(* IEC 61131-3 sources: brOscatLib/oscatNetw (part 3) *)

(* ---- HTTP_GET.st ---- *)
FUNCTION_BLOCK HTTP_GET
    (*http://www.oscat.de/images/OSCATNetwork/oscat_netlib121_en.pdf#page=98*)
    CASE state OF
    00:	DONE := FALSE;
    	IF GET AND NOT get_last THEN (* auf positive Flanke SET warten *)
    		state := 10;
    		ip4_stored := IP4; (* aktuelle IP4 speichern *)
    		total_size := 0;
    		HEADER_START := UINT#0;
    		HEADER_STOP := UINT#0;
    		BODY_START := UINT#0;
    		BODY_STOP := UINT#0;
    		HTTP_STATUS := '';
    		ERROR := DWORD#0;
    		ip_state := BYTE#1; (* Anmelden *)
    		authentication := FALSE;
    		delimiter2b := '$0D$0A';
    		delimiter4b := '$0D$0A$0D$0A';

    		(* LOGIN Parameter vorhanden *)
    		(* LOGIN Parameter vorhanden *)
    		IF URL_DATA.USER <> '' AND URL_DATA.PASSWORD <> '' THEN
    			b64_str1 := CONCAT(URL_DATA.USER,':');
    			b64_str1 := CONCAT(b64_str1,URL_DATA.PASSWORD); (* USER:PASSWORD *)
    			b64_start := TRUE; (* BASE64 kodierung von Username *)
    			authentication := TRUE;
    			state := 5;
    		ELSE
    			state := 10;
    		END_IF
    	        	(*####################  DEBUG-MESSAGE  ###################################*)
    		(*IF _debug_enable THEN
    	       		LOG_CL.NEW_MSG := 'HTTP: S00 START /ip_id ~4';
    	            	LOG_CL.PRINTF[4]  := BYTE_TO_STRING(ip_id);
    	            	LOG_MSG();
    	        	END_IF*)
    	        	(*########################################################################*)
    	END_IF

    5:	IF b64_start AND b64_done THEN (* warten auf base64 konvertierung *)
    		b64_start := FALSE;
    		state := 10;
    	END_IF

    10:	IF ip_state = BYTE#3 THEN (* Bei IP_Control anmelden und auf freigabe warten *)
    		idx := 0;
    		text := CONCAT('GET ',URL_DATA.PATH);
    		_STRING_TO_BUFFER(STR:=text,POS:=idx,PT:=ADR(S_BUF.BUFFER),SIZE:=SIZEOF(S_BUF.BUFFER)); (* GET path in buffer kopieren *)
    		idx := idx + LEN(text);

    		IF LEN(URL_DATA.QUERY) > 0 THEN
    			S_BUF.BUFFER[idx] := 63; (* ASCII '?' *)
    			idx := idx + 1;
    			_STRING_TO_BUFFER(STR:=URL_DATA.QUERY,POS:=idx,PT:=ADR(S_BUF.BUFFER),SIZE:=SIZEOF(S_BUF.BUFFER)); (* QUERY in buffer kopieren *)
    			idx := idx + LEN(URL_DATA.QUERY);
    		END_IF

    		IF MODE >= BYTE#2 THEN (* gewünschte HTTP Version uebergeben *)
    			text := ' HTTP/1.1';
    		ELSE
    			text := ' HTTP/1.0';
    		END_IF
    		text := CONCAT(text,delimiter2b);
    		_STRING_TO_BUFFER(STR:=text,POS:=idx,PT:=ADR(S_BUF.BUFFER),SIZE:=SIZEOF(S_BUF.BUFFER)); (* HTTP Version in buffer kopieren *)
    		idx := idx + LEN(text);

    		IF MODE = BYTE#1 THEN (* HTTP/1.0 mit persistenter Verbindung gewünscht *)
    			text := CONCAT('Connection: Keep-Alive',delimiter2b); (* workaround für pcworx -> kein $0D$0A als Stringkonstante möglich *)
    		ELSIF MODE = BYTE#3 THEN (* HTTP/1.1 ohne persistenter Verbindung gewünscht *)
    			text := CONCAT('Connection: Close',delimiter2b); (* workaround für pcworx -> kein $0D$0A als Stringkonstante möglich *)
    		ELSE
    			text := '';
    		END_IF

    		(* Zusatz Parameter übernehmen *)
    		text := CONCAT(text,URL_DATA.HEADER);
    		_STRING_TO_BUFFER(STR:=text,POS:=idx,PT:=ADR(S_BUF.BUFFER),SIZE:=SIZEOF(S_BUF.BUFFER)); (* HTTP Version in buffer kopieren *)
    		idx := idx + LEN(text);

    		IF authentication THEN
    			text := CONCAT('Authorization: Basic ',b64_str2);
    			text := CONCAT(text,delimiter2b); (* workaround für pcworx -> kein $0D$0A als Stringkonstante möglich *)
    			_STRING_TO_BUFFER(STR:=text,POS:=idx,PT:=ADR(S_BUF.BUFFER),SIZE:=SIZEOF(S_BUF.BUFFER)); (* HTTP Host in buffer kopieren *)
    			idx := idx + LEN(text);
    		END_IF

    		text := CONCAT('Host: ',URL_DATA.DOMAIN);
    		text := CONCAT(text,delimiter4b); (* workaround für pcworx -> kein $0D$0A als Stringkonstante möglich *)
    		_STRING_TO_BUFFER(STR:=text,POS:=idx,PT:=ADR(S_BUF.BUFFER),SIZE:=SIZEOF(S_BUF.BUFFER)); (* HTTP Host in buffer kopieren *)
    		idx := idx + LEN(text);

    		(* IP Datenverkehr einrichten *)
    		IF FIND(';HTTPS;https;Https;', CONCAT(URL_DATA.PROTOCOL,';')) > 1 THEN
    			IP_C.C_PORT := SEL(URL_DATA.PORT = WORD#0,URL_DATA.PORT,WORD#443); (* Portnummer eintragen *)
    			IP_C.MAILBOX[16] := BYTE#1; (* SSL MODE freigeben *)
    		ELSE
    			IP_C.C_PORT := SEL(URL_DATA.PORT = WORD#0,URL_DATA.PORT,WORD#80);  (* Portnummer eintragen *)
    		END_IF

    		IP_C.C_IP := ip4_stored; (* IP eintragen *)
    		IP_C.C_MODE := BYTE#0; (* MODE: TCP+AKTIV+PORT+IP *)
    		IP_C.C_ENABLE := TRUE; (* Verbindungsaufbau freigeben *)
    		IP_C.TIME_RESET := TRUE; (* Zeitueberwachung rücksetzen *)
    		IP_C.R_OBSERVE := TRUE; (* Datenempfang ueberwachen *)
    		S_BUF.SIZE := INT_TO_UINT(idx); (* Sendelänge eintragen *)
    		R_BUF.SIZE := UINT#0; (* Empfangslänge rücksetzen *)

    		state := 30;
    	        	(*####################  DEBUG-MESSAGE  ###################################*)
    	        	(*IF _debug_enable THEN
    	        		LOG_CL.NEW_MSG := 'HTTP: S20 SEND /ip_id ~4';
    	            	LOG_CL.PRINTF[4]  := BYTE_TO_STRING(ip_id);
    	            	LOG_MSG();
    	        	END_IF*)
    	        	(*########################################################################*)
    	END_IF

    30:	rcv_timeout := (IP_C.ERROR AND DWORD#16#0000_FF00) = DWORD#16#0000_FF00;
    	con_rdce :=     (IP_C.ERROR AND DWORD#16#FD00_0000) = DWORD#16#FD00_0000;

    	IF S_BUF.SIZE = UINT#0 THEN
    		IF total_size = 0 THEN
    			IF R_BUF.SIZE > UINT#15 THEN; (* länge der empfangenen Daten prüfen *)

    				(* HTTP HEADER Ende suchen -> durch $0D$A$0D$A erkennbar bei DEC RT-11,CP/M,MS-DOS,Windows *)
    				del_end := '$0D$0A$0D$0A';
    				del_pos := BUFFER_SEARCH(PT:=ADR(R_BUF.BUFFER),SIZE:=R_BUF.SIZE,STR:=del_end,POS:=0,IGN:=FALSE);

    				(* kein Ende gefunden ? -> andere Ende-Codierung suchen *)
    				IF del_pos = 0 THEN
    					del_end := '$0A$0A';
    					(* HTTP HEADER Ende suchen -> durch $0A$0A erkennbar bei Multics, Unix-Derivate,Mac OS X *)
    					del_pos := BUFFER_SEARCH(PT:=ADR(R_BUF.BUFFER),SIZE:=R_BUF.SIZE,STR:=del_end,POS:=0,IGN:=FALSE);
    				END_IF

    				IF del_pos > 0 THEN
    					HEADER_START := UINT#0;
    					HEADER_STOP := INT_TO_UINT(del_pos + LEN(del_end) - 1);
    					total_size := -1; (* HTTP Header empfangen aber noch keine gesamtlänge bekannt *)
    				END_IF
    		                	(*####################  DEBUG-MESSAGE  ###################################*)
    		                	(*IF _debug_enable THEN
    		                   	LOG_CL.NEW_MSG := 'HTTP: S20 HEADER_START ~1 / HEADER_STOP ~2/ip_id ~4';
    		                   	LOG_CL.PRINTF[4]  := BYTE_TO_STRING(ip_id);
    		                   	LOG_CL.PRINTF[1]  := UINT_TO_STRING(HEADER_START);
    		                   	LOG_CL.PRINTF[2]  := UINT_TO_STRING(HEADER_STOP);
    		                   	LOG_MSG();
    		                	END_IF*)
    		                	(*########################################################################*)

    				(* HTTP Statuscode auswerten: (kann 1.0 oder 1.1 sein *)
    				READ_HTTP(size:=HEADER_STOP,pos:=0,SRC:='',pt:=R_BUF.BUFFER);

    				i := LEN(READ_HTTP.READ_HTTP);
    				IF i > 7 THEN
    					(* HTTP Version von HOST auswerten 1.0 oder 1.1 *)
    					text:=MID(READ_HTTP.READ_HTTP,1,3);
    					http_1_1_host := text = '1';

    					(* Code und Meldung isolieren *)
    					HTTP_STATUS := RIGHT(READ_HTTP.READ_HTTP,i-4);
    				END_IF

    				(* positive HTTP Anfrage ? *)
    				IF FIND(HTTP_STATUS,'200') > 0 THEN

    					(* 'Content-Length: Wert einlesen auswerten *)
    					READ_HTTP(size:=HEADER_STOP,pos:=0,SRC:='CONTENT-LENGTH',pt:=R_BUF.BUFFER);
    					text:=READ_HTTP.READ_HTTP;

    					IF LEN(text) >= 1 THEN
    						IF IS_NUM(str:=text) THEN
    							(* erwartete gesamtmenge an Bytes berechnen *)
    							total_size := STRING_TO_INT(text) + UINT_TO_INT(HEADER_STOP) + 1;
                               					(*####################  DEBUG-MESSAGE  ###################################*)
                               					(*IF _debug_enable THEN
                                  					LOG_CL.NEW_MSG := 'HTTP: S20 HEADER ~1, BODY ~2 TOTAL ~3 /ip_id ~4';
                                 					LOG_CL.PRINTF[4]  := BYTE_TO_STRING(ip_id);
                                   					LOG_CL.PRINTF[1]  := UINT_TO_STRING(HEADER_STOP);
                                   					LOG_CL.PRINTF[2]  := INT_TO_STRING(total_size-UINT_TO_INT(HEADER_STOP));
                                   					LOG_CL.PRINTF[3]  := INT_TO_STRING(total_size);
                                  					LOG_MSG();
                              					END_IF*)
                              					(*########################################################################*)
    						END_IF
    					END_IF
    				ELSE
    					ERROR := DWORD#16#000000FC; (* Fehler durch HTTP-Statuscodes *)
    				END_IF
    			END_IF
    		(* 1. bei bekannter Content-Length wird nach erhalt der erwartenen Daten die verbindung beendet *)
    		(* 2. bei persistenter Verbindung muss bei unbekannter Datenmenge auf Receive-Timeout gewartet werden *)
    		(* 3. wenn nach datenempfang die verbindung vom host unterbrochen wird *)
    		ELSIF (R_BUF.SIZE >= INT_TO_UINT(total_size)) OR
    			(R_BUF.SIZE > UINT#0 AND total_size < 0 AND ((rcv_timeout OR con_rdce) OR (IP_C.C_STATE = BYTE#1))) THEN

    			IF R_BUF.SIZE - 1 > HEADER_STOP THEN (* BODY Daten vorhanden *)
    				BODY_START := HEADER_STOP + UINT#1;
    				BODY_STOP := R_BUF.SIZE - 1;
    		                	(*####################  DEBUG-MESSAGE  ###################################*)
    		                	(*IF _debug_enable THEN
    		                   	LOG_CL.NEW_MSG := 'HTTP: S20 BODY ~1, START ~2 END ~3 /ip_id ~4';
    		                   	LOG_CL.PRINTF[4]  := BYTE_TO_STRING(ip_id);
    		                   	LOG_CL.PRINTF[1]  := UINT_TO_STRING(HEADER_STOP);
    		                   	LOG_CL.PRINTF[2]  := UINT_TO_STRING(BODY_START);
    		                   	LOG_CL.PRINTF[3]  := UINT_TO_STRING(BODY_STOP);
    		                   	LOG_MSG();
    		               	END_IF*)
    		               	(*########################################################################*)
    			END_IF

    			DONE := TRUE;
    			IP_C.C_ENABLE := FALSE; (* Verbindung abbauen *)
    			state := 40;
                		(*####################  DEBUG-MESSAGE  ###################################*)
                		(*IF _debug_enable THEN
                    			LOG_CL.NEW_MSG := 'HTTP: S30 OK /ip_id ~4';
                    			LOG_CL.PRINTF[4]  := BYTE_TO_STRING(ip_id);
                    			LOG_MSG();
                		END_IF*)
                		(*########################################################################*)
    		END_IF
    	END_IF

    	IF IP_C.ERROR <> DWORD#0 THEN
    		(* bei unbekannter Content-size ist nicht bekannt ob bzw wieviele Telegramme noch folgen werden *)
    		(* darum wird nach receive-timeout oder Remote disconnect ERROR der fehler wieder ausgefiltert (logischer fehler) *)
    		IF rcv_timeout AND DONE THEN
    			IP_C.ERROR := IP_C.ERROR AND DWORD#16#FFFF_00FF; (* Fehler wieder rücksetzen *)
    		ELSIF con_rdce AND DONE THEN
    			IP_C.ERROR := IP_C.ERROR AND DWORD#16#00FF_FFFF; (* Fehler wieder rücksetzen *)
    		ELSE
    			ERROR := IP_C.ERROR;
    		END_IF
    	END_IF

    	IF ERROR > DWORD#0 THEN
    		IP_C.C_ENABLE := FALSE; (* Verbindungsaufbau sperren *)
    		state := 40;
    	        	(*####################  DEBUG-MESSAGE  ###################################*)
    	        	(*IF _debug_enable THEN
    	            	LOG_CL.NEW_MSG := 'HTTP: S30 ERROR ~1 /ip_id ~4';
    	            	LOG_CL.PRINTF[1]  := DWORD_TO_STRING(ERROR);
    	            	LOG_CL.PRINTF[4]  := BYTE_TO_STRING(ip_id);
    	            	LOG_MSG();
    	        	END_IF*)
    	        	(*########################################################################*)
    	END_IF

    40:	IF (UNLOCK_BUF OR NOT DONE) THEN (* Warten auf Release und Verbindung beendet -> ip_id vom Stack nehmen *)
    		ip_state := BYTE#4; (* Abmelden *)
    		DONE := FALSE;
    		IP_C.MAILBOX[16] := BYTE#0; (* SSL MODE beenden *)
    		state := 0;
    	END_IF
    END_CASE

    get_last := GET; (* letzten Status sichern zur Flankenerkennung *)

    IP_FIFO(FIFO:=IP_C.FIFO,state:=ip_state,ID:=ip_id); (* IP_FIFO *)

    BASE64_ENCODE_STR(RUN:=b64_start,STR1:=b64_str1,STR2:=b64_str2); (* BASE64 kodierung *)
    b64_done:=BASE64_ENCODE_STR.DONE;

    (*####################  DEBUG-MESSAGE  ###################################*)
    (*IF _debug_enable THEN
    	IF state <> _debug_state_last THEN
    		LOG_CL.NEW_MSG := 'http_get: /last ~1 /New ~2';
    		LOG_CL.PRINTF[1] := INT_TO_STRING(_debug_state_last);
    		LOG_CL.PRINTF[2] := INT_TO_STRING(state);
    		LOG_MSG();
    		_debug_state_last := state;
    	END_IF
    END_IF*)
    (*########################################################################*)

    (* revision history
    ks	18. oct. 2008	rev 1.0
    	original version

    ks	20. oct. 2009	rev 1.1
    	Fehler bei body-suche bei $0a$0a korrigiert,Codeoptimierung,
    	new VAR del_pos , del_end (Networkbuffer und Buffer-funktionen auf Basis 0)

    ks	28. oct. 2009	rev 1.2
    	über url.header können zusätzliche header-infos übergeben werden

    ks	12. apr. 2011	rev 1.3
    	verbesserte fehlererkennung und fehlerkorrektur bei buffer_to_string

    ks	31. mar. 2016	rev 1.4
    	authentication und SSL (HTTPS) hinzugefügt, DONE später zurücksetzen

    *)
END_FUNCTION_BLOCK

(* ---- INI_PARSER_BUF.st ---- *)
FUNCTION_BLOCK INI_PARSER_BUF
    (*http://www.oscat.de/images/OSCATNetwork/oscat_netlib121_en.pdf#page=161*)
    IF RUN > 0 THEN
    	IF state = 0 THEN (* Auswertung neu beginnen *)

    		pv := ADR(VALUE);
    		pv := 0; (* VALUE = '' *)
    		pve := pv + INT_TO_DWORD(STRING_LENGTH);
    		pk := ADR(KEY);
    		pk := 0; (* KEY = '' *)
    		pke := pk + INT_TO_DWORD(STRING_LENGTH);

    		i := UDINT_TO_INT(OFFSET);
    		size := UINT_TO_INT(PT.size) - 1;
    		RESULT := 0;
    		state := 5; (* Befehl in Arbeit (Busy) *)
    		step := 0; (* Auswertung neu beginnen *)

    		(*####################  DEBUG-MESSAGE  ###################################*)
    		(*IF _debug_enable THEN
    			LOG_CL.NEW_MSG := 'IPB: Startindex: ~1';
    			LOG_CL.PRINTF[1]  := INT_TO_STRING(i);
    			LOG_MSG();
    		END_IF*)
    		(*########################################################################*)
    	END_IF

    	watchdog(IN:=FALSE,PT:=T#1ms); (* Timer neustarten *)
    	watchdog.IN := TRUE;

    	WHILE (state = 5) DO (* Schleife solange kein Ergebnis *)

    		watchdog(); (* Timer aktualisieren *)

    		IF watchdog.Q THEN (* watchdog ausgelöst *)
    			state := 5;
    			EXIT;
    		ELSIF i > size THEN (* kein weiteres zeichen vorhanden *)
    			state := 10; (* nichts gefunden - Daten-Ende erreicht *)
    			EXIT;
    		ELSE

    			c := PT.BUFFER[i]; (* neues Zeichen aus Buffer lesen *)
    			eof := i + 1 = PT.size; (* End of File *)

    			k_add := 0;
    			v_add := 0;

    			CASE step OF

    			0: (* noch kein Modus erkannt *)
    				IF c = 91 THEN (* mit "[" vergleichen *)
    					step := 200; (* Modus für Section aktivieren *)
    				ELSIF c = 59 OR c = 35 THEN (* mit ";" und '#' vergleichen *)
    					step := 100; (* Modus für Kommentar aktivieren *)
    				ELSIF c > 32 THEN (* KEY erkannt *)
    					k_add := c; (* Zeichen ablegen *)
    					step := 300; (* KEY auswertung starten *)
    				END_IF
    			100: (* Kommentar erkannt -> Zeilenende suchen *)
    				IF c < 32 THEN (* prüfe auf Steuerzeichen *)
    					state  := 3; (* Beenden -> Kommentar wurde gefunden *)
    				END_IF
    			200: (* Sections-start erkannt -> Sectionsende suchen *)
    				IF c = 93 THEN (* mit "]" vergleichen *)
    					IF pk > ADR(KEY) > 0 THEN (* innerhalb von [] muss sich mindestens ein Zeichen befinden *)
    						state  := 1; (* Beenden -> Section wurde gefunden *)
    					ELSE
    						pk := ADR(KEY);
    						pk := 0; (* KEY = '' *)
    						step := 0; (* fehlerhafte Section-Zeile vorhanden -> weitersuchen *)
    					END_IF
    				ELSIF c < 32 OR eof THEN (* Steuerzeichen - fehlerhafte Section-Zeile -> weitersuchen *)
    					pk := ADR(KEY);
    					pk := 0; (* KEY = '' *)
    					step := 0;
    				ELSE
    					k_add := c; (* Zeichen ablegen *)
    				END_IF
    			300: (* Beginn: KEY erkannt -> Name auswerten *)
    				IF c < 32 THEN (* Steuerzeichen - fehlerhafte KEY-Zeile -> weitersuchen *)
    					pk := ADR(KEY);
    					pk := 0; (* KEY = '' *)
    					step := 0;
    				ELSIF c = 61 THEN (* prüfe auf '=' *)
    					step := 330;
    				ELSE
    					k_add := c; (* Zeichen ablegen *)
    				END_IF
    			330: (* KeyValue beginn suchen *)
    				IF c < 32 THEN (* Steuerzeichen  *)
    					state := 2; (* KEY ohne VALUE gefunden *)
    				ELSIF eof THEN
    					state := 2; (* KEY ohne VALUE gefunden *)
    					v_add := c; (* Zeichen ablegen *)
    				ELSE
    					v_add := c; (* Zeichen ablegen *)
    					step := 350;
    				END_IF
    			350: (* KeyValue Ende suchen *)
    				IF c < 32 THEN (* Steuerzeichen *)
    					state := 2; (* KEY gefunden *)
    				ELSIF eof THEN
    					v_add := c; (* Zeichen ablegen *)
    					state := 2; (* KEY gefunden *)
    				ELSE
    					v_add := c; (* Zeichen ablegen *)
    				END_IF
    			END_CASE

    			IF v_add > 0  AND pv < pve THEN (* Zeichen zu VALUE-String hinzufügen *)
    				pv := v_add; (* Zeichen eintragen *)
    				pv := pv + 1;
    				pv := 0; (* String-Terminierung eintragen *)
    			END_IF

    			IF k_add > 0 AND pk < pke THEN (* Zeichen zu KEY-String hinzufügen *)
    				pk := k_add; (* Zeichen eintragen *)
    				pk := pk + 1;
    				pk := 0; (* String-Terminierung eintragen *)
    			END_IF

    			i := i + 1; (* Datenzeiger erhöhen *)

    		END_IF
    	END_WHILE

    	CASE state OF
    	01:	(* Section gefunden *)
    		IF RUN = 1 OR RUN = 3 THEN (* Section vorgewählt oder alles rückmelden *)
    			IF KEY = STR OR LEN(STR) = 0 THEN (* mit gesuchter Section vergleichen oder keine Section vorgegeben *)
    				RESULT := 1; (* Section gefunden *)
    				OFFSET := i; (* OFFSET uebernehmen *)
    				RUN := 0;
    				state := 0;
    			END_IF
    		ELSE
    			pk := ADR(KEY);
    			pk := 0; (* KEY = '' *)
    			RESULT := 11; (* KEY nicht gefunden , Section-Ende - OFFSET nicht verändern *)
    			RUN := 0;
    			state := 0;
    		END_IF
    	02:	(* KEY gefunden *)
    		IF RUN = 2 OR RUN = 3 THEN (* KEY vorgewählt oder alles rückmelden *)
    			IF KEY = STR OR LEN(STR) = 0 THEN (* mit gesuchten KEY vergleichen *)
    				RESULT := 2; (* KEY gefunden *)
    				OFFSET := i; (* OFFSET uebernehmen *)
    				RUN := 0;
    				state := 0;
    			END_IF
    		END_IF
    	03:	(* Kommenar gefunden *)
    		OFFSET := i; (* OFFSET uebernehmen *)
    		state := 0;

    	05:	RESULT := 5; (* in Arbeit *)

    	10:	(* Indexüberschreitung - Bufferende *)
    		RESULT := 10; (* nichts gefunden - Datenende erreicht *)
    		OFFSET := i; (* OFFSET uebernehmen *)
    		RUN := 0;
    		state := 0;
    	END_CASE

    	(*####################  DEBUG-MESSAGE  ###################################*)
    	(*IF _debug_enable THEN
    		LOG_CL.NEW_MSG := 'IPF: intern RESULT ~1 , state ~2, step ~3 , OFFSET ~4, RUN ~5';
    		LOG_CL.PRINTF[1] := BYTE_TO_STRING(RESULT);
    		LOG_CL.PRINTF[2] := BYTE_TO_STRING(state);
    		LOG_CL.PRINTF[3] := INT_TO_STRING(step);
    		LOG_CL.PRINTF[4] := UDINT_TO_STRING(OFFSET);
    		LOG_CL.PRINTF[5] := BYTE_TO_STRING(RUN);
    		LOG_MSG();
    	END_IF*)
    	(*########################################################################*)

    END_IF

    (*####################  DEBUG-MESSAGE  ###################################*)
    (*IF _debug_enable THEN
    	IF step_last <> step THEN
    		LOG_CL.NEW_MSG := 'IPB: step: ~1';
    		LOG_CL.PRINTF[1]  := INT_TO_STRING(step);
    		LOG_MSG();
    	END_IF
    	step_last := step;
    END_IF*)
    (*########################################################################*)

    (* revision history
    ks	23. sep. 2010	rev 1.0
    	original version
    *)
END_FUNCTION_BLOCK

(* ---- INI_PARSER_FILE.st ---- *)
FUNCTION_BLOCK INI_PARSER_FILE
    (*http://www.oscat.de/images/OSCATNetwork/oscat_netlib121_en.pdf#page=164*)
    IF RUN > 0 THEN

    	IF state = 0 THEN (* Auswertung neu beginnen *)
    		pv := ADR(VALUE);
    		pv := 0; (* VALUE = '' *)
    		pve := pv + INT_TO_DWORD(STRING_LENGTH);
    		pk := ADR(KEY);
    		pk := 0; (* KEY = '' *)
    		pke := pk + INT_TO_DWORD(STRING_LENGTH);

    		i := OFFSET;
    		RESULT := 0;
    		state := 5; (* Befehl in Arbeit (Busy) *)
    		step := 0; (* Auswertung neu beginnen *)

    		(*####################  DEBUG-MESSAGE  ###################################*)
    		(*IF _debug_enable THEN
    			LOG_CL.NEW_MSG := 'IPF: Startindex: ~1';
    			LOG_CL.PRINTF[1] := UDINT_TO_STRING(i);
    			LOG_MSG();
    		END_IF*)
    		(*########################################################################*)

    	END_IF

    	watchdog(IN:=FALSE,PT:=T#1ms); (* Timer neustarten *)
    	watchdog.IN := TRUE;

    	WHILE (state = 5) DO (* Schleife solange kein Ergebnis *)

    		mode := 1;
    		FB(mode:=mode,FSD:=FSD,PT:=PT,FILENAME:=FILENAME,POS:=i );
    		e:=FB.ERROR;
    		c:=FB.DATA;

    		eof := i + 1 = FSD.FILE_SIZE; (* End of File *)

    		(*####################  DEBUG-MESSAGE  ###################################*)
    		(*IF _debug_enable THEN
    			LOG_CL.NEW_MSG := 'IPF: mode: ~1, error: ~2 , >~7<>~3< ~4 step ~5 index ~6';
    			LOG_CL.PRINTF[1] := BYTE_TO_STRING(mode);
    			LOG_CL.PRINTF[2] := BYTE_TO_STRING(e);
    			LOG_CL.PRINTF[3] := BYTE_TO_STRING(c);
    			LOG_CL.PRINTF[4] := BOOL_TO_STRING(eof);
    			LOG_CL.PRINTF[5] := INT_TO_STRING(step);
    			LOG_CL.PRINTF[6] := UDINT_TO_STRING(i);
    			LOG_CL.PRINTF[7] := CHR_TO_STRING(c);
    			LOG_MSG();
    		END_IF*)
    		(*########################################################################*)

    		watchdog(); (* Timer aktualisieren *)

    		IF mode > 0 OR watchdog.Q THEN (* Baustein noch aktiv, oder watchdog ausgelöst *)
    			state := 5;
    			EXIT;
    		ELSIF e > 0 THEN (* File_error oder kein weiteres zeichen vorhanden *)
    			state := 10; (* nichts gefunden - Daten-Ende erreicht *)
    			EXIT;
    		ELSE

    			k_add := 0;
    			v_add := 0;

    			CASE step OF

    			0: (* noch kein Modus erkannt *)
    				IF c = 91 THEN (* mit "[" vergleichen *)
    					step := 200; (* Modus für Section aktivieren *)
    				ELSIF c = 59 OR c = 35 THEN (* mit ";" und '#' vergleichen *)
    					step := 100; (* Modus für Kommentar aktivieren *)
    				ELSIF c > 32 THEN (* KEY erkannt *)
    					k_add := c; (* Zeichen ablegen *)
    					step := 300; (* KEY auswertung starten *)
    				END_IF
    			100: (* Kommentar erkannt -> Zeilenende suchen *)
    				IF c < 32 THEN (* prüfe auf Steuerzeichen *)
    					state  := 3; (* Beenden -> Kommentar wurde gefunden *)
    				END_IF
    			200: (* Sections-start erkannt -> Sectionsende suchen *)
    				IF c = 93 THEN (* mit "]" vergleichen *)
    					IF pk > ADR(KEY) > 0 THEN (* innerhalb von [] muss sich mindestens ein Zeichen befinden *)
    						state  := 1; (* Beenden -> Section wurde gefunden *)
    					ELSE
    						pk := ADR(KEY);
    						pk := 0; (* KEY = '' *)
    						step := 0; (* fehlerhafte Section-Zeile vorhanden -> weitersuchen *)
    					END_IF
    				ELSIF c < 32 OR eof THEN (* Steuerzeichen - fehlerhafte Section-Zeile -> weitersuchen *)
    					pk := ADR(KEY);
    					pk := 0; (* KEY = '' *)
    					step := 0;
    				ELSE
    					k_add := c; (* Zeichen ablegen *)
    				END_IF
    			300: (* Beginn: KEY erkannt -> Name auswerten *)
    				IF c < 32 THEN (* Steuerzeichen - fehlerhafte KEY-Zeile -> weitersuchen *)
    					pk := ADR(KEY);
    					pk := 0; (* KEY = '' *)
    					step := 0;
    				ELSIF c = 61 THEN (* prüfe auf '=' *)
    					step := 330;
    				ELSE
    					k_add := c; (* Zeichen ablegen *)
    				END_IF
    			330: (* KeyValue beginn suchen *)
    				IF c < 32 THEN (* Steuerzeichen  *)
    					state := 2; (* KEY ohne VALUE gefunden *)
    				ELSIF eof THEN
    					state := 2; (* KEY ohne VALUE gefunden *)
    					v_add := c; (* Zeichen ablegen *)
    				ELSE
    					v_add := c; (* Zeichen ablegen *)
    					step := 350;
    				END_IF
    			350: (* KeyValue Ende suchen *)
    				IF c < 32 THEN (* Steuerzeichen *)
    					state := 2; (* KEY gefunden *)
    				ELSIF eof THEN
    					v_add := c; (* Zeichen ablegen *)
    					state := 2; (* KEY gefunden *)
    				ELSE
    					v_add := c; (* Zeichen ablegen *)
    				END_IF
    			END_CASE

    			IF v_add > 0  AND pv < pve THEN (* Zeichen zu VALUE-String hinzufügen *)
    				pv := v_add; (* Zeichen eintragen *)
    				pv := pv + 1;
    				pv := 0; (* String-Terminierung eintragen *)
    			END_IF

    			IF k_add > 0 AND pk < pke THEN (* Zeichen zu KEY-String hinzufügen *)
    				pk := k_add; (* Zeichen eintragen *)
    				pk := pk + 1;
    				pk := 0; (* String-Terminierung eintragen *)
    			END_IF

    			i := i + 1; (* Datenzeiger erhöhen *)

    		END_IF
    	END_WHILE

    	CASE state OF
    	01:	(* Section gefunden *)
    		IF RUN = 1 OR RUN = 3 THEN (* Section vorgewählt oder alles rückmelden *)
    			IF KEY = STR OR LEN(STR) = 0 THEN (* mit gesuchter Section vergleichen oder keine Section vorgegeben *)
    				RESULT := 1; (* Section gefunden *)
    				OFFSET := i; (* OFFSET uebernehmen *)
    				RUN := 0;
    				state := 0;
    			END_IF
    		ELSE
    			pk := ADR(KEY);
    			pk := 0; (* KEY = '' *)
    			RESULT := 11; (* KEY nicht gefunden , Section-Ende - OFFSET nicht verändern *)
    			RUN := 0;
    			state := 0;
    		END_IF
    	02:	(* KEY gefunden *)
    		IF RUN = 2 OR RUN = 3 THEN (* KEY vorgewählt oder alles rückmelden *)
    			IF KEY = STR OR LEN(STR) = 0 THEN (* mit gesuchten KEY vergleichen *)
    				RESULT := 2; (* KEY gefunden *)
    				OFFSET := i; (* OFFSET uebernehmen *)
    				RUN := 0;
    				state := 0;
    			END_IF
    		END_IF
    	03:	(* Kommenar gefunden *)
    		OFFSET := i; (* OFFSET uebernehmen *)
    		state := 0;

    	05:	RESULT := 5; (* in Arbeit *)

    	10:	(* Indexüberschreitung - Bufferende *)
    		RESULT := 10; (* nichts gefunden - Datenende erreicht *)
    		OFFSET := i; (* OFFSET uebernehmen *)
    		RUN := 0;
    		state := 0;
    	END_CASE

    	(*####################  DEBUG-MESSAGE  ###################################*)
    	(*IF _debug_enable THEN
    		LOG_CL.NEW_MSG := 'IPF: intern RESULT ~1 , state ~2, step ~3 , OFFSET ~4, RUN ~5';
    		LOG_CL.PRINTF[1] := BYTE_TO_STRING(RESULT);
    		LOG_CL.PRINTF[2] := BYTE_TO_STRING(state);
    		LOG_CL.PRINTF[3] := INT_TO_STRING(step);
    		LOG_CL.PRINTF[4] := UDINT_TO_STRING(OFFSET);
    		LOG_CL.PRINTF[5] := BYTE_TO_STRING(RUN);
    		LOG_MSG();
    	END_IF*)
    	(*########################################################################*)

    END_IF

    (*####################  DEBUG-MESSAGE  ###################################*)
    (*IF _debug_enable THEN
    	IF step_last <> step THEN
    		LOG_CL.NEW_MSG := 'IPB: step: ~1';
    		LOG_CL.PRINTF[1]  := INT_TO_STRING(step);
    		LOG_MSG();
    	END_IF
    	step_last := step;
    END_IF*)
    (*########################################################################*)

    (* revision history
    ks	23. sep. 2010	rev 1.0
    	original version
    *)
END_FUNCTION_BLOCK

(* ---- IP2GEO.st ---- *)
FUNCTION_BLOCK IP2GEO
    (*http://www.oscat.de/images/OSCATNetwork/oscat_netlib121_en.pdf#page=99*)
    CASE state OF

    00:
    	IF ACTIVATE AND NOT last_state THEN
    		state := 20;
    		DONE := FALSE;
    		BUSY := TRUE;
    		ERROR_C := DWORD#0;
    		ERROR_T := BYTE#0;
    	END_IF

    20: (* URL for DNS UND HTTP-GET *)
    	(* Example: http://ipinfodb.com/ip_query.php?IP=10.10.10.10 *)
    	(* Example: http://ipinfodb.com/ip_query.php?timezone=true&IP=*)
    	URL_DATA:=STRING_TO_URL(STR:='http://ipinfodb.com/ip_query.php?timezone=true&IP=',DEFAULT_PROTOCOL:='',DEFAULT_PATH:='');

    	IF IP > DWORD#0 THEN
    		URL_DATA.QUERY := CONCAT(URL_DATA.QUERY,IP4_TO_STRING(IP4:=IP));
    	END_IF

    	state := 40;

    40:
    	IF DNS_CLIENT.DONE THEN
    		state := 60;
    	ELSIF (DNS_CLIENT.ERROR > DWORD#00) THEN
    		(* Fehlerbehandlung *)
    		ERROR_C := DNS_CLIENT.ERROR;
    		ERROR_T := BYTE#01;
    		state := 100;
    	END_IF

    60:
    	IF HTTP_GET.DONE THEN
    		state := 80;
    		CTRL.START_POS := HTTP_GET.BODY_START;
    		CTRL.STOP_POS := HTTP_GET.BODY_STOP;
    		CTRL.COMMAND := WORD#2#10000000_00011000; (* ONLY TEXT AND ATTRIBUTE *)
    		CTRL.WATCHDOG := T#1ms;

    	ELSIF (HTTP_GET.ERROR > DWORD#00) THEN
    		(* Fehlerbehandlung *)
    		ERROR_C := HTTP_GET.ERROR;
    		ERROR_T := BYTE#02;
    		state := 100;
    	END_IF

    80:
    	(* XML Daten seriell lesen *)
    	XML_READER(CTRL:=CTRL,BUF:=R_BUF.BUFFER);
    	IF CTRL.TYP < 98 THEN (* nur auswerten wenn kein Watchdog durchlauf *)
    		(* automatische konvertierung in real und int ausführen *)
    		value_int := 0;
    		value_real := 0.0;
    		IF LEN(CTRL.VALUE) <= 20 THEN
    			v_real :=FLOAT_TO_REAL(FLT:=CTRL.VALUE);
    			IF CHK_REAL(v_real) = 0 THEN (* !!! prüft auf gültigen REAL Wert, ansonsten stürzt Twincat ab !!!!  *)
    				value_real := v_real;
    				value_int := REAL_TO_INT(value_real);
    			END_IF
    		END_IF

    		CASE UINT_TO_INT(CTRL.COUNT) OF

    		07: GEO.IP4 := IP4_DECODE(STR:=CTRL.VALUE); (* IP-Adresse *)
    		10: GEO.state := 'OK' = CTRL.VALUE; (* STATUS *)
    		13: GEO.COUNTRY_CODE := CTRL.VALUE; (* Country-Code *)
    		16: GEO.COUNTRY_NAME := CTRL.VALUE; (* Country-Name *)
    		19: GEO.REGION_CODE := CTRL.VALUE; (* Region-Code *)
    		22: GEO.REGION_NAME := CTRL.VALUE; (* Region-Name *)
    		25: GEO.CITY := CTRL.VALUE; (* City *)
    		31: GEO.GEO_LATITUDE := value_real; (* Latitude *)
    		34: GEO.GEO_LONGITUDE := value_real; (* Longitude *)
    		37: GEO.TIME_ZONE_NAME := CTRL.VALUE; (* TimeZone Name *)
    		40: GEO.GMT_OFFSET := value_int; (* GMT OFFSET in Sekunden *)
    		43: GEO.IS_DST := value_int > 0; (* Sommerzeit aktiv *)
    		END_CASE

    	ELSIF CTRL.TYP = 99 THEN (* EXIT - letztes Element gelesen *)
    		DONE := TRUE;
    		state := 100;
    	END_IF

    100:
    	(* UNLOCK HTTP DATA *)
    	IF (NOT HTTP_GET.DONE) THEN
    		state := 0;
    		BUSY := FALSE;
    		DONE := ERROR_T = BYTE#0;
    	END_IF

    END_CASE

    (* ---------------- DNS --------------- *)
    DNS_CLIENT(	IP_C:=IP_C,
    			S_BUF:=S_BUF,
    			R_BUF:=R_BUF,
    			DOMAIN:=URL_DATA.DOMAIN,
    			IP4_DNS:=DWORD#00,
    			ACTIVATE:=state=40 (* DNS Start *)
    			);

    (* nicht oder nicht direkt verwendete Parameter *)
    (* 	DWORD :=DNS_CLIENT.IP4;
    	BOOL  :=DNS_CLIENT.DONE;
    	BYTE  :=DNS_CLIENT.ERROR; *)
    (* -------------------------------------*)

    (* ------------- HTTP_GET --------------- *)
    HTTP_GET(	IP_C:=IP_C,
    			S_BUF:=S_BUF,
    			R_BUF:=R_BUF,
    			IP4:=DNS_CLIENT.IP4,
    			GET:=state=60,
    			MODE:=BYTE#2, (* HTTP 1.1 mit persistenter Verbindung *)
    			UNLOCK_BUF:=state=100,
    			URL_DATA:=URL_DATA
    			);

    (* nicht oder nicht direkt verwendete Parameter *)
    (*	STRING := HTTP_GET.HTTP_STATUS;
    	UINT :=HTTP_GET.HEADER_START;
    	UINT :=HTTP_GET.HEADER_STOP;
    	UINT :=HTTP_GET.BODY_START;
    	UINT :=HTTP_GET.BODY_STOP;
    	BOOL :=HTTP_GET.DONE;
    	BYTE :=HTTP_GET.ERROR;
    *)
    (* -------------------------------------*)

    last_state := ACTIVATE;

    (* revision history
    ks	14. aug. 2009	rev 1.0
    	original version

    ks	07. oct. 2010	rev 1.1
    	new url , ip2geo fields , REAL_CHECK
    *)
END_FUNCTION_BLOCK

(* ---- IP_CONTROL.st ---- *)
FUNCTION_BLOCK IP_CONTROL
    (*http://www.oscat.de/images/OSCATNetwork/oscat_netlib121_en.pdf#page=101*)
    (* ---------------------- Debug-Message ----------------------------*)
    (*IF _debug_enable THEN
    	IF IP_C.FIFO.ID > BYTE#0 THEN
    		debug_index := IP_C.FIFO.NR;
    		debug_ID := BYTE_TO_INT(IP_C.FIFO.X[debug_index]);
    	END_IF
    END_IF*)
    (* -----------------------------------------------------------------------------*)

    (* read system time *)
    tx := T_PLC_MS();

    IF IP_C.c_port = 0 THEN
    	IP_C.c_port := PORT; (* uebergebenen PORT durch parametrierten PORT ersetzen *)
    END_IF
    IF IP_C.c_ip = 0 AND IP_C.c_mode < 4 THEN
    	IP_C.c_ip := IP; (* uebergebene IP durch paramtrierte IP ersetzen *)
    END_IF

    new_connection := c_ip <> IP_C.c_ip OR c_mode <> IP_C.c_mode OR c_port <> IP_C.c_port; (* neue Verbindungs erwünscht ? *)
    c_enable := IP_C.c_enable AND NOT new_connection;

    IF IP_C.c_enable AND IP_C.ERROR = 0 AND state = STOP THEN (* Freigabe,kein Fehler,kein socket offen *)
    	c_ip   := IP_C.c_ip;
    	c_mode := IP_C.c_mode;
    	c_port := IP_C.c_port;
    	plc_841 := SYSLIBSOCKETS_OPTION.1; (* Bit 1 = WAGO 750-841 *)
    	plc_881 := SYSLIBSOCKETS_OPTION.2; (* Bit 1 = WAGO 750-881 *)
    	udp_mode := c_mode.0; (* Mode 1,3,5 = udp *)

    	error_time := TIME_TO_DWORD(MAX(T#200ms,TIME_OUT));
    	IP_C.TIME_RESET := TRUE; (* Alle Timer ruecksetzen *)

    	r_max_size := SIZEOF(R_BUF.BUFFER);
    	s_max_size := SIZEOF(S_BUF.BUFFER);

    	IF c_mode.0 THEN (* Mode: 1,3,5 = UDP CLIENT/SERVER *)
    		state := UDP_INIT;
    	ELSIF c_mode = 0 THEN (* Mode: 0 = TCP CLIENT *)
    		state := TC_INIT;
    	ELSE
    		state := TS_INIT; (* Mode: 2,4 = TCP SERVER *)
    	END_IF

    	(* ---------------------- Debug-Message ----------------------------*)
    	(*IF _debug_enable THEN
    		LOG_CL.NEW_MSG := 'IP_CON: MODE ~1 / IP ~2 / PORT ~3 /ID ~6';
    		LOG_CL.PRINTF[1] := BYTE_TO_STRING(c_mode);
    		LOG_CL.PRINTF[2] := IP4_TO_STRING(c_ip);
    		LOG_CL.PRINTF[3] := WORD_TO_STRING(c_port);
    		LOG_CL.PRINTF[6] := INT_TO_STRING(debug_ID);
    		LOG_MSG();
    	END_IF*)
    	(* -----------------------------------------------------------------------------*)

    END_IF

    (* ---------------------- Debug-Message ----------------------------*)
    (*IF  _debug_enable THEN
    	IF state <> state_last THEN
    		LOG_CL.NEW_MSG := 'IP_STEP ~1 -IP_ID ~6';
    		LOG_CL.PRINTF[1] := BYTE_TO_STRING(state);
    		LOG_CL.PRINTF[6] := INT_TO_STRING(debug_ID);
    		LOG_MSG();
    		state_last := state;
    	END_IF
    END_IF*)
    (* -----------------------------------------------------------------------------*)

    IF IP_C.TIME_RESET THEN (* Alle Timer ruecksetzen *)
    	IP_C.TIME_RESET := FALSE; (* Reset rücksetzen *)
    	c_time := tx; (* Connect Timer ruecksetzen *)
    	s_time := tx; (* Send Timer ruecksetzen *)
    	r_time := tx; (* Receive Timer ruecksetzen *)

    	c_status := BYTE#0; (* letzten Connect Fehler rücksetzen *)
    	s_status := BYTE#0; (* letzten Send Fehler rücksetzen *)
    	r_status := BYTE#0; (* letzten Receive Fehler rücksetzen *)
    END_IF

    (* ---------------------------------------------- *)

    CASE state OF

    UDP_INIT: (* UDP_CLIENT + SERVER *)
    	socket := SysSockCreate(SOCKET_AF_INET, SOCKET_DGRAM, SOCKET_IPPROTO_IP);
    	IF socket < 0 THEN
    		c_status := 1; (* SysSockCreate failed *)
    		state := C_CLOSE;
    	ELSE
    		SysSockSetOption(socket, SOCKET_SOL, SOCKET_SO_BROADCAST, ADR(dint_true), SIZEOF(dint_true)); (* allow broadcast *)
    		SysSockIoctl(socket, SOCKET_FIONBIO, ADR(dint_true)); (* put socket in non-blocking mode *)
    		sockaddr.sin_family := SOCKET_AF_INET;
    		sockaddr.sin_port := SysSockHtons(c_port);
    		sockaddr.sin_addr := SEL(c_mode = 1, SOCKET_INADDR_ANY, SysSockNtohl(c_ip));

    		IF c_mode >= 2 THEN (* SERVER Mode *)
    			IF SysSockBind(socket, ADR(sockaddr), SIZEOF(sockaddr)) THEN
    				c_ready := TRUE; (* Connected *)
    				state:= C_WAIT;
    			ELSE
    				c_status := 2; (* SysSockBind failed *)
    				state := C_CLOSE;
    			END_IF
    		ELSE
    			c_ready := TRUE; (* Connected *)
    			state:= C_WAIT;
    		END_IF
    	END_IF

    (* ---------------------------------------------- *)

    TC_INIT: (* TCP-CLIENT (AKTIV) *)
    	socket := SysSockCreate(SOCKET_AF_INET, SOCKET_STREAM, SOCKET_IPPROTO_IP);
    	IF socket < 0 THEN
    		c_status := 1;  (* SysSockCreate failed *)
    		state := C_CLOSE;
    	ELSE
    		IF plc_841 OR plc_881 THEN
    			SysSockSetOption(socket,6,SOCKET_TCP_NODELAY, ADR(dint_true), SIZEOF(dint_true)); (* Set Push-Bit *)
    		END_IF
    		SysSockIoctl(socket, SOCKET_FIONBIO, ADR(dint_true)); (* NonBlocking mode *)
    		sockaddr.sin_family := SOCKET_AF_INET;
    		sockaddr.sin_port := SysSockNtohs(c_port);
    		sockaddr.sin_addr := SysSockNtohl(c_ip);
    		c_select := FALSE;
    		state := TC_CONNECT;
    	END_IF

    (* ---------------------------------------------- *)

    TC_CONNECT:
    	IF NOT c_enable OR c_status = 255 THEN (* keine freigabe oder connect timeout *)
    			state:= C_CLOSE;
    	ELSE
    		IF c_select = FALSE THEN
    			IF SysSockConnect(socket,ADR(sockaddr),SIZEOF(sockaddr)) THEN
    				c_ready := TRUE; (* Connected *)
    				state:= C_WAIT;
    			ELSE
    				(* Connect durchgeführt, aber noch nicht verbunden, dann optional mit select-abfrage weitermachen *)
    				c_select := SYSLIBSOCKETS_OPTION.0; (* Bit 0 = TCP-Client - use SysSockselect *)
    			END_IF
    		ELSE
    			c_Timeout.tv_sec := 0;
    			c_Timeout.tv_usec := 0;
    			c_fdWrite.fd_count := 1;
    			c_fdWrite.fd_array[0] := socket;
    			IF SysSockSelect(SOCKET_FD_SETSIZE,0,ADR(c_fdWrite),0, ADR(c_Timeout)) > 0 THEN
    				c_ready := TRUE; (* Connected *)
    				state:= C_WAIT;
    			END_IF
    		END_IF
    	END_IF

    (* ---------------------------------------------- *)

    TS_INIT: (* TCP-SERVER (PASSIV) *)
    	server_socket := SysSockCreate(SOCKET_AF_INET, SOCKET_STREAM, SOCKET_IPPROTO_IP); (* Create socket *)
    	IF server_socket = SOCKET_INVALID THEN
    		c_status := 1; (* SysSockCreate failed *)
    		state:= C_CLOSE;
    	ELSE (* Address bindings *)
    		SysSockSetOption( server_socket, SOCKET_SOL, SOCKET_SO_REUSEADDR, ADR(dint_true), SIZEOF(dint_true) );
    		sockaddr.sin_family:= SOCKET_AF_INET;
    		sockaddr.sin_port := SysSockHtons(c_port);
    		sockaddr.sin_addr := SOCKET_INADDR_ANY;
    		IF NOT SysSockBind(server_socket, ADR(sockaddr), SIZEOF(sockaddr)) THEN
    			c_status := 2; (* SysSockBind failed *)
    			state := C_CLOSE;
    		ELSIF NOT SysSockListen(server_socket, 1) THEN (* erzeugt Warteschlange für eine Verbindung *)
    			c_status := 3; (* SysSockListen failed *)
    			state:= C_CLOSE;
    		ELSE
    			SysSockIoctl(server_socket, SOCKET_FIONBIO, ADR(dint_true)); (* NonBlocking mode *)
    			state:= TS_OPEN;
    		END_IF
    	END_IF

    (* ---------------------------------------------- *)

    TS_OPEN: (* Waiting for incomming connection *)
    	sockaddr_size := SIZEOF(sockaddr);
    	socket := SysSockAccept(server_socket, ADR(sockaddr), ADR(sockaddr_size));

    	IF socket <> SOCKET_INVALID THEN (* neuer Verbindungswunsch vorhanden *)
    		IF c_mode = BYTE#2 AND sockaddr.sin_addr <> SysSockNtohl(c_ip) THEN (* Mode 2 = TCP + PASSIVE + PORT + IP  auf richtige Partner-IP prüfen *)
    			state:= C_CLOSE;
    		ELSE
    			IF plc_841 OR plc_881 THEN
    				SysSockSetOption(socket, 6, SOCKET_TCP_NODELAY, ADR(dint_true), SIZEOF(dint_true)); (* Set Push-Bit *)
    			END_IF
    			SysSockIoctl(socket, SOCKET_FIONBIO, ADR(dint_true)); (* NonBlocking mode *)
    			c_ready := TRUE; (* Connected *)
    			state := C_WAIT;
    		END_IF
    	ELSIF NOT c_enable THEN (* keine freigabe mehr ? *)
    			state:= C_CLOSE;
    	END_IF

    (* ---------------------------------------------- *)

    C_WAIT: (* Warten auf Anforderung für Beenden *)
    	IF NOT c_enable OR NOT c_ready THEN
    		state:= C_CLOSE;
    	END_IF

    (* ---------------------------------------------- *)

    C_CLOSE: (* Close the Sockets *)
    	c_ready := FALSE;
    	IF socket >= 0 THEN
    		IF (NOT plc_841) AND (NOT plc_881) THEN
    			SysSockShutdown(socket, 0); (* 870 *)
    		END_IF
    		SysSockClose(socket);
    		socket := SOCKET_INVALID;
    	END_IF
    	IF server_socket >= 0 THEN
    		IF (NOT plc_841) AND (NOT plc_881) THEN
    			SysSockShutdown(server_socket, 0); (* 870 *)
    		END_IF
    		SysSockClose(server_socket);
    		server_socket := SOCKET_INVALID;
    	END_IF
    	state:= STOP;
    END_CASE

    (* ---------------------------------------------- *)

    IF c_ready THEN
    	IF NOT c_ready_old THEN (* Verbindung aufgebaut - positive Flanke erkannt *)
    		IP_C.C_STATE := 254;
    		IP_C.TIME_RESET := TRUE; (* Alle Timer ruecksetzen *)
    		(* ---------------------- Debug-Message ----------------------------*)
    		(*IF _debug_enable THEN
    			LOG_CL.NEW_MSG := 'IP_CON: CONNECTED -IP_ID ~6';
    			LOG_CL.PRINTF[6] := INT_TO_STRING(debug_ID);
    			LOG_MSG();
    		END_IF*)
    		(* -----------------------------------------------------------------------------*)
    	ELSE
    		IP_C.C_STATE := 255; (* Verbindung ist aufgebaut *)
    	END_IF
    ELSE
    	IF c_ready_old THEN (* Verbindung abgebaut - negative Flanke erkannt *)
    		IP_C.C_STATE := 1;
    		IP_C.MAILBOX[1] := 0; (* Receive Info rücksetzen *)
    		IP_C.MAILBOX[2] := 0; (* Send-Pause rücksetzen *)
    		IP_C.MAILBOX[3] := 0; (* Receive-Pause rücksetzen *)
    		IF NOT new_connection THEN
    			s_active := FALSE; (* Sendeaktivitäten stoppen *)
    			s_req := FALSE; (* Sendefreigabe rücksetzen *)
    			S_BUF.SIZE := 0; (* Sendelänge löschen *)
    			(*IP_C.TIME_RESET := TRUE;*) (* Alle Timer ruecksetzen *)
    		END_IF
    		(* ---------------------- Debug-Message ----------------------------*)
    		(*IF _debug_enable THEN
    			LOG_CL.NEW_MSG := 'IP_CON: DISCONNECTED';
    			LOG_MSG();
    		END_IF*)
    		(* -----------------------------------------------------------------------------*)
    	ELSE
    		IP_C.C_STATE := 0; (* Verbindung ist abgebaut *)
    	END_IF
    END_IF

    c_ready_old := c_ready;

    (* Der Datenempfang wird angehalten solange ein Sendevorgang läuft *)
    (* sonst kann es vorkommen das die Antwort-daten schon empfangen werden, *)
    (* bevor der Sendevorgang vom programm abgeschlossen wurde *)

    IF c_ready AND NOT s_active AND IP_C.MAILBOX[3] = 0 THEN
    	IF R_BUF.SIZE >= INT_TO_UINT(r_max_size) THEN
    		R_BUF.SIZE := UINT#0;
    		r_status := 254; (* Empfangsbuffer wegen Überlauf rückgesetzt *)
    	END_IF

    	r_offset := SEL(udp_mode,UINT_TO_INT(R_BUF.SIZE),0);
    	r_count := r_max_size - r_offset;

    	IF udp_mode THEN
    		bytes_received := SysSockRecvFrom(socket, ADR(R_BUF.BUFFER), r_count, 0, ADR(sockaddr), SIZEOF(sockaddr));

    		IF c_mode = BYTE#3 AND sockaddr.sin_addr <> SysSockNtohl(c_ip) THEN (* Mode 3 = UDP + PASSIVE + PORT + IP  auf richtige Partner-IP prüfen *)
    			bytes_received := 0;
    			R_BUF.SIZE := UINT#0;
    			sockaddr.sin_port := SysSockNtohs(c_port);
    			sockaddr.sin_addr := SysSockNtohl(c_ip);
    		END_IF

    	ELSE
    		bytes_received := SysSockRecv(socket, ADR(R_BUF.BUFFER[r_offset]), r_count, 0);
    	END_IF

    	(*UDP: IPC returns -1 if no data available or error occured,841 returns -1 if error occured and 0 if no data available*)
    	CASE bytes_received OF
    	-2147483648..-1: ; (* No data available or error occured *)
    	 0: IF NOT udp_mode THEN (* TCP-Mode: socket wurde von remote geschlossen *)
    			c_status := 253;
    			c_ready := FALSE;
    		END_IF
    	ELSE (* daten wurden empfangen *)
      		r_time := tx; (* Receive Timer ruecksetzen *)
    		R_BUF.SIZE := INT_TO_UINT(r_offset + DINT_TO_UINT(bytes_received)); (* aktuelle buffersize eintragen *)
    		IP_C.MAILBOX[1] := IP_C.MAILBOX[1] + 1; (* Receive Info *)
    		IF IP_C.MAILBOX[1] = 0 THEN IP_C.MAILBOX[1] := 1; END_IF

    		(* ---------------------- Debug-Message ----------------------------*)
    		(*IF _debug_enable THEN
    			LOG_CL.NEW_MSG := 'IP_REC DATA: POS: ~1 : SIZE: ~2 TOTAL ~3 -IP_ID ~6';
    			LOG_CL.PRINTF[1] := INT_TO_STRING(r_offset);
    			LOG_CL.PRINTF[2] := INT_TO_STRING(r_count);
    			LOG_CL.PRINTF[3] := UINT_TO_STRING(R_BUF.SIZE);
    			LOG_CL.PRINTF[6] := INT_TO_STRING(debug_ID);
    			LOG_MSG();
    		END_IF*)
    		(* -----------------------------------------------------------------------------*)

    	END_CASE
    END_IF

    (* ---------------------------------------------- *)

    IF S_BUF.SIZE > 0 THEN
    	IF c_ready AND c_enable THEN
    		IF NOT s_active AND IP_C.MAILBOX[2] = 0 THEN
    			(* Gesamtanzahl an Bytes limitieren und uebergeben *)
    			s_total := LIMIT(0,UINT_TO_INT(S_BUF.SIZE),r_max_size);
    			s_cur_pos  := 0;
    			s_cur_size := 0;
    			s_start := TRUE; (* Daten kopieren und senden anstossen *)
    			s_active := TRUE; (* Sende-Betrieb aktivieren *)
    			(* ---------------------- Debug-Message ----------------------------*)
    			(*IF _debug_enable THEN
    				LOG_CL.NEW_MSG := 'IP_SEN INIT: TOTAL: ~1 -IP_ID ~6';
    				LOG_CL.PRINTF[1] := INT_TO_STRING(s_total);
    				LOG_CL.PRINTF[6] := INT_TO_STRING(debug_ID);
    				LOG_MSG();
    			END_IF*)
    			(* -----------------------------------------------------------------------------*)
    		END_IF

    		IF s_done OR s_start THEN (* Daten senden aktiv *)

    			s_start := FALSE;
    			s_cur_pos := s_cur_pos + s_cur_size; (* neue Sende-Datenposition bestimmen *)
    			IF s_total > s_cur_pos THEN (* weitere Daten zum senden vorhanden ? *)
    				s_cur_size := s_total - s_cur_pos;
    				s_cur_size := LIMIT(0, s_cur_size, s_max_size); (* Telegrammlänge begrenzen *)
    				(* ---------------------- Debug-Message ----------------------------*)
    				(*IF _debug_enable THEN
    					LOG_CL.NEW_MSG := 'IP_SEN DATA: POS: ~1 : SIZE: ~2 TOTAL ~3 -IP_ID ~6';
    					LOG_CL.PRINTF[1] := INT_TO_STRING(s_cur_pos);
    					LOG_CL.PRINTF[2] := INT_TO_STRING(s_cur_size);
    					LOG_CL.PRINTF[3] := INT_TO_STRING(s_total);
    					LOG_CL.PRINTF[6] := INT_TO_STRING(debug_ID);
    					LOG_MSG();
    				END_IF*)
    				(* -----------------------------------------------------------------------------*)
    				s_time := tx; (* Send Timer ruecksetzen *)
    				r_time := tx; (* Receive Timer ruecksetzen *)
    				s_req := TRUE;

    			ELSE
    				(* keine weitere Sendedaten vorhanden -> Senden beenden *)
    				s_req := FALSE;
    				s_active := FALSE;
    				S_BUF.SIZE := 0;
    				(* ---------------------- Debug-Message ----------------------------*)
    				(*IF _debug_enable THEN
    					LOG_CL.NEW_MSG := 'IP_SEN FINISH -IP_ID ~6';
    					LOG_CL.PRINTF[6] := INT_TO_STRING(debug_ID);
    					LOG_MSG();
    				END_IF*)
    				(* -----------------------------------------------------------------------------*)
    			END_IF
    		END_IF
    	END_IF
    END_IF

    IF s_req THEN
    	s_done := FALSE;
    	IF udp_mode THEN
    		bytes_sent := SysSockSendTo(socket, ADR(S_BUF.BUFFER[s_cur_pos]), s_cur_size, 0, ADR(sockaddr), SIZEOF(sockaddr));
    	ELSE
    		bytes_sent := SysSockSend(socket, ADR(S_BUF.BUFFER[s_cur_pos]), s_cur_size, 0);
    	END_IF

    	CASE bytes_sent OF
    	-2147483648..-1:	; (* ERROR: Noch nicht bereit um Daten aufzunehmen -> nächsten Zyklus wieder probieren *)
    	 0: IF NOT udp_mode THEN (* TCP-Mode: socket wurde von remote geschlossen *)
    			c_status := 253;
    			c_ready := FALSE;
    		END_IF
    	ELSE
    		s_done := TRUE;
    		s_cur_size := DINT_TO_INT(bytes_sent); (* Anzahl der wirklich versendeten Bytes übernehmen *)
    		(* ---------------------- Debug-Message ----------------------------*)
    		(*IF _debug_enable THEN
    			LOG_CL.NEW_MSG := 'IP_SEN SEND_COUNT ~1 -IP_ID ~6';
    			LOG_CL.PRINTF[1] := DINT_TO_STRING(s_cur_size);
    			LOG_CL.PRINTF[6] := INT_TO_STRING(debug_ID);
    			LOG_MSG();
    		END_IF*)
    		(* -----------------------------------------------------------------------------*)
    	END_CASE
    END_IF

    (* ---------------------------------------------- *)

    IF IP_C.R_OBSERVE = FALSE OR s_active THEN
        r_time := tx;
    END_IF

    IF c_status = 0 AND tx - c_time > error_time AND c_enable AND NOT c_ready AND c_mode < 2 THEN (* Connect Timeout *)
    	c_status := 255; (* Timeout-Fehler ausgeben *)
    END_IF
    IF s_status = 0 AND tx - s_time > error_time AND s_active THEN (* Send Timeout *)
    	s_status := 255; (* Timeout-Fehler ausgeben *)
    END_IF
    IF r_status = 0 AND tx - r_time > error_time AND c_ready AND IP_C.R_OBSERVE THEN (* Receive Timeout *)
    	r_status := 255; (* Timeout-Fehler ausgeben *)
    END_IF

    IP_C.ERROR := DWORD_OF_BYTE(c_status,s_status,r_status,0);

    (* ---------------------- Debug-Message ----------------------------*)
    (*IF  _debug_enable THEN
    	IF (IP_C.ERROR <> debug_lasterror) THEN
    		LOG_CL.NEW_MSG := 'IP_ERROR ~1 -IP_ID ~6';
    		LOG_CL.PRINTF[1] := DWORD_TO_STRING(IP_C.ERROR);
    		LOG_CL.PRINTF[6] := INT_TO_STRING(debug_ID);
    		LOG_MSG();

    		debug_lasterror := IP_C.ERROR;
    		debug_last_id := debug_ID;
    	END_IF
    END_IF*)
    (* -----------------------------------------------------------------------------*)

    (* revision history
    ks	18. oct. 2008	rev 1.0
    	original version
    ks	05. jan. 2009	rev 1.1
    	zusätzlichen Parameter "PORT" hinzugefügt, und Code bei Verbindungsaufbau angepasst
    ks	28. feb. 2009	rev 1.2
    	connect code angepasst und verkürzung der zyklen bei Send
    ks	20. oct. 2009	rev 1.3
    	network_buffer basis 0
    ks	06. dec. 2009	rev 1.4
    	receive_count MAILBOX[1]
    ks	10. nov. 2010	rev 1.5
    	send_pause MAILBOX[2] and receive_pause MAILBOX[3]
    ks	07. feb. 2011	rev 1.6
    	Fehlercode 253 bei Remote-Verbindungsabbruch
    ks	30. may. 2011	rev 1.7
    	Fehler bei Empfangsüberwachung
    ks	26. july. 2011	rev 1.8
    	Error-Reset, diverse optimierungen
    ks	26. feb. 2012	rev 1.9
    	Code-Optimierung für höhere kompatibilität

    *)
END_FUNCTION_BLOCK

(* ---- IP_CONTROL2.st ---- *)
FUNCTION_BLOCK IP_CONTROL2
    (*http://www.oscat.de/images/OSCATNetwork/oscat_netlib121_en.pdf#page=107*)
    (* ---------------------- Debug-Message ----------------------------*)
    (*IF _debug_enable THEN
    	IF IP_C.FIFO.ID > BYTE#0 THEN
    		debug_index := IP_C.FIFO.NR;
    		debug_ID := BYTE_TO_INT(IP_C.FIFO.X[debug_index]);
    	END_IF
    END_IF*)
    (* -----------------------------------------------------------------------------*)

    (* read system time *)
    tx := T_PLC_MS();

    IF IP_C.c_port = 0 THEN
    	IP_C.c_port := PORT; (* uebergebenen PORT durch parametrierten PORT ersetzen *)
    END_IF
    IF IP_C.c_ip = 0 AND IP_C.c_mode < 4 THEN
    	IP_C.c_ip := IP; (* uebergebene IP durch paramtrierte IP ersetzen *)
    END_IF

    new_connection := c_ip <> IP_C.c_ip OR c_mode <> IP_C.c_mode OR c_port <> IP_C.c_port; (* neue Verbindungs erwünscht ? *)
    c_enable := IP_C.c_enable AND NOT new_connection;

    IF IP_C.c_enable AND IP_C.ERROR = 0 AND state = STOP THEN (* Freigabe,kein Fehler,kein socket offen *)
    	c_ip   := IP_C.c_ip;
    	c_mode := IP_C.c_mode;
    	c_port := IP_C.c_port;
    	plc_841 := SYSLIBSOCKETS_OPTION.1; (* Bit 1 = WAGO 750-841 *)
    	plc_881 := SYSLIBSOCKETS_OPTION.2; (* Bit 1 = WAGO 750-881 *)
    	udp_mode := c_mode.0; (* Mode 1,3,5 = udp *)

    	error_time := TIME_TO_DWORD(MAX(T#200ms,TIME_OUT));
    	IP_C.TIME_RESET := TRUE; (* Alle Timer ruecksetzen *)

    	r_max_size := SIZEOF(R_BUF.BUFFER);
    	s_max_size := SIZEOF(S_BUF.BUFFER);

    	IF c_mode.0 THEN (* Mode: 1,3,5 = UDP CLIENT/SERVER *)
    		state := UDP_INIT;
    	ELSIF c_mode = 0 THEN (* Mode: 0 = TCP CLIENT *)
    		state := TC_INIT;
    	ELSE
    		state := TS_INIT; (* Mode: 2,4 = TCP SERVER *)
    	END_IF

    	(* ---------------------- Debug-Message ----------------------------*)
    	(*IF _debug_enable THEN
    		LOG_CL.NEW_MSG := 'IP_CON: MODE ~1 / IP ~2 / PORT ~3 /ID ~6';
    		LOG_CL.PRINTF[1] := BYTE_TO_STRING(c_mode);
    		LOG_CL.PRINTF[2] := IP4_TO_STRING(c_ip);
    		LOG_CL.PRINTF[3] := WORD_TO_STRING(c_port);
    		LOG_CL.PRINTF[6] := INT_TO_STRING(debug_ID);
    		LOG_MSG();
    	END_IF*)
    	(* -----------------------------------------------------------------------------*)

    END_IF

    (* ---------------------- Debug-Message ----------------------------*)
    (*IF  _debug_enable THEN
    	IF state <> state_last THEN
    		LOG_CL.NEW_MSG := 'IP_STEP ~1 -IP_ID ~6';
    		LOG_CL.PRINTF[1] := BYTE_TO_STRING(state);
    		LOG_CL.PRINTF[6] := INT_TO_STRING(debug_ID);
    		LOG_MSG();
    		state_last := state;
    	END_IF
    END_IF*)
    (* -----------------------------------------------------------------------------*)

    IF IP_C.TIME_RESET THEN (* Alle Timer ruecksetzen *)
    	IP_C.TIME_RESET := FALSE; (* Reset rücksetzen *)
    	c_time := tx; (* Connect Timer ruecksetzen *)
    	s_time := tx; (* Send Timer ruecksetzen *)
    	r_time := tx; (* Receive Timer ruecksetzen *)

    	c_status := BYTE#0; (* letzten Connect Fehler rücksetzen *)
    	s_status := BYTE#0; (* letzten Send Fehler rücksetzen *)
    	r_status := BYTE#0; (* letzten Receive Fehler rücksetzen *)
    END_IF

    (* ---------------------------------------------- *)

    CASE state OF

    UDP_INIT: (* UDP_CLIENT + SERVER *)
    	socket := SysSockCreate(SOCKET_AF_INET, SOCKET_DGRAM, SOCKET_IPPROTO_IP);
    	IF socket < 0 THEN
    		c_status := 1; (* SysSockCreate failed *)
    		state := C_CLOSE;
    	ELSE
    		SysSockSetOption(socket, SOCKET_SOL, SOCKET_SO_BROADCAST, ADR(dint_true), SIZEOF(dint_true)); (* allow broadcast *)
    		SysSockIoctl(socket, SOCKET_FIONBIO, ADR(dint_true)); (* put socket in non-blocking mode *)
    		sockaddr.sin_family := SOCKET_AF_INET;
    		sockaddr.sin_port := SysSockHtons(c_port);
    		sockaddr.sin_addr := SEL(c_mode = 1, SOCKET_INADDR_ANY, SysSockNtohl(c_ip));

    		IF c_mode >= 2 THEN (* SERVER Mode *)
    			IF SysSockBind(socket, ADR(sockaddr), SIZEOF(sockaddr)) THEN
    				c_ready := TRUE; (* Connected *)
    				state:= C_WAIT;
    			ELSE
    				c_status := 2; (* SysSockBind failed *)
    				state := C_CLOSE;
    			END_IF
    		ELSE
    			c_ready := TRUE; (* Connected *)
    			state:= C_WAIT;
    		END_IF
    	END_IF

    (* ---------------------------------------------- *)

    TC_INIT: (* TCP-CLIENT (AKTIV) *)
    	socket := SysSockCreate(SOCKET_AF_INET, SOCKET_STREAM, SOCKET_IPPROTO_IP);
    	IF socket < 0 THEN
    		c_status := 1;  (* SysSockCreate failed *)
    		state := C_CLOSE;
    	ELSE
    		IF plc_841 OR plc_881 THEN
    			SysSockSetOption(socket,6,SOCKET_TCP_NODELAY, ADR(dint_true), SIZEOF(dint_true)); (* Set Push-Bit *)
    		END_IF
    		SysSockIoctl(socket, SOCKET_FIONBIO, ADR(dint_true)); (* NonBlocking mode *)
    		sockaddr.sin_family := SOCKET_AF_INET;
    		sockaddr.sin_port := SysSockNtohs(c_port);
    		sockaddr.sin_addr := SysSockNtohl(c_ip);
    		c_select := FALSE;
    		state := TC_CONNECT;
    	END_IF

    (* ---------------------------------------------- *)

    TC_CONNECT:
    	IF NOT c_enable OR c_status = 255 THEN (* keine freigabe oder connect timeout *)
    			state:= C_CLOSE;
    	ELSE
    		IF c_select = FALSE THEN
    			IF SysSockConnect(socket,ADR(sockaddr),SIZEOF(sockaddr)) THEN
    				c_ready := TRUE; (* Connected *)
    				state:= C_WAIT;
    			ELSE
    				(* Connect durchgeführt, aber noch nicht verbunden, dann optional mit select-abfrage weitermachen *)
    				c_select := SYSLIBSOCKETS_OPTION.0; (* Bit 0 = TCP-Client - use SysSockselect *)
    			END_IF
    		ELSE
    			c_Timeout.tv_sec := 0;
    			c_Timeout.tv_usec := 0;
    			c_fdWrite.fd_count := 1;
    			c_fdWrite.fd_array[0] := socket;
    			IF SysSockSelect(SOCKET_FD_SETSIZE,0,ADR(c_fdWrite),0, ADR(c_Timeout)) > 0 THEN
    				c_ready := TRUE; (* Connected *)
    				state:= C_WAIT;
    			END_IF
    		END_IF
    	END_IF

    (* ---------------------------------------------- *)

    TS_INIT: (* TCP-SERVER (PASSIV) *)
    	server_socket := SysSockCreate(SOCKET_AF_INET, SOCKET_STREAM, SOCKET_IPPROTO_IP); (* Create socket *)
    	IF server_socket = SOCKET_INVALID THEN
    		c_status := 1; (* SysSockCreate failed *)
    		state:= C_CLOSE;
    	ELSE (* Address bindings *)
    		SysSockSetOption( server_socket, SOCKET_SOL, SOCKET_SO_REUSEADDR, ADR(dint_true), SIZEOF(dint_true) );
    		sockaddr.sin_family:= SOCKET_AF_INET;
    		sockaddr.sin_port := SysSockHtons(c_port);
    		sockaddr.sin_addr := SOCKET_INADDR_ANY;
    		IF NOT SysSockBind(server_socket, ADR(sockaddr), SIZEOF(sockaddr)) THEN
    			c_status := 2; (* SysSockBind failed *)
    			state := C_CLOSE;
    		ELSIF NOT SysSockListen(server_socket, 1) THEN (* erzeugt Warteschlange für eine Verbindung *)
    			c_status := 3; (* SysSockListen failed *)
    			state:= C_CLOSE;
    		ELSE
    			SysSockIoctl(server_socket, SOCKET_FIONBIO, ADR(dint_true)); (* NonBlocking mode *)
    			state:= TS_OPEN;
    		END_IF
    	END_IF

    (* ---------------------------------------------- *)

    TS_OPEN: (* Waiting for incomming connection *)
    	sockaddr_size := SIZEOF(sockaddr);
    	socket := SysSockAccept(server_socket, ADR(sockaddr), ADR(sockaddr_size));

    	IF socket <> SOCKET_INVALID THEN (* neuer Verbindungswunsch vorhanden *)
    		IF c_mode = BYTE#2 AND sockaddr.sin_addr <> SysSockNtohl(c_ip) THEN (* Mode 2 = TCP + PASSIVE + PORT + IP  auf richtige Partner-IP prüfen *)
    			state:= C_CLOSE;
    		ELSE
    			IF plc_841 OR plc_881 THEN
    				SysSockSetOption(socket, 6, SOCKET_TCP_NODELAY, ADR(dint_true), SIZEOF(dint_true)); (* Set Push-Bit *)
    			END_IF
    			SysSockIoctl(socket, SOCKET_FIONBIO, ADR(dint_true)); (* NonBlocking mode *)
    			c_ready := TRUE; (* Connected *)
    			state := C_WAIT;
    		END_IF
    	ELSIF NOT c_enable THEN (* keine freigabe mehr ? *)
    			state:= C_CLOSE;
    	END_IF

    (* ---------------------------------------------- *)

    C_WAIT: (* Warten auf Anforderung für Beenden *)
    	IF NOT c_enable OR NOT c_ready THEN
    		state:= C_CLOSE;
    	END_IF

    (* ---------------------------------------------- *)

    C_CLOSE: (* Close the Sockets *)
    	c_ready := FALSE;
    	IF socket >= 0 THEN
    		IF (NOT plc_841) AND (NOT plc_881) THEN
    			SysSockShutdown(socket, 0); (* 870 *)
    		END_IF
    		SysSockClose(socket);
    		socket := SOCKET_INVALID;
    	END_IF
    	IF server_socket >= 0 THEN
    		IF (NOT plc_841) AND (NOT plc_881) THEN
    			SysSockShutdown(server_socket, 0); (* 870 *)
    		END_IF
    		SysSockClose(server_socket);
    		server_socket := SOCKET_INVALID;
    	END_IF
    	state:= STOP;
    END_CASE

    (* ---------------------------------------------- *)

    IF c_ready THEN
    	IF NOT c_ready_old THEN (* Verbindung aufgebaut - positive Flanke erkannt *)
    		IP_C.C_STATE := 254;
    		IP_C.TIME_RESET := TRUE; (* Alle Timer ruecksetzen *)
    		(* ---------------------- Debug-Message ----------------------------*)
    		(*IF _debug_enable THEN
    			LOG_CL.NEW_MSG := 'IP_CON: CONNECTED -IP_ID ~6';
    			LOG_CL.PRINTF[6] := INT_TO_STRING(debug_ID);
    			LOG_MSG();
    		END_IF*)
    		(* -----------------------------------------------------------------------------*)
    	ELSE
    		IP_C.C_STATE := 255; (* Verbindung ist aufgebaut *)
    	END_IF
    ELSE
    	IF c_ready_old THEN (* Verbindung abgebaut - negative Flanke erkannt *)
    		IP_C.C_STATE := 1;
    		IP_C.MAILBOX[1] := 0; (* Receive Info rücksetzen *)
    		IP_C.MAILBOX[2] := 0; (* Send-Pause rücksetzen *)
    		IP_C.MAILBOX[3] := 0; (* Receive-Pause rücksetzen *)
    		IF NOT new_connection THEN
    			s_active := FALSE; (* Sendeaktivitäten stoppen *)
    			s_req := FALSE; (* Sendefreigabe rücksetzen *)
    			S_BUF.SIZE := 0; (* Sendelänge löschen *)
    			(* IP_C.TIME_RESET := TRUE; *) (* Alle Timer ruecksetzen *)
    		END_IF
    		(* ---------------------- Debug-Message ----------------------------*)
    		(*IF _debug_enable THEN
    			LOG_CL.NEW_MSG := 'IP_CON: DISCONNECTED';
    			LOG_MSG();
    		END_IF*)
    		(* -----------------------------------------------------------------------------*)
    	ELSE
    		IP_C.C_STATE := 0; (* Verbindung ist abgebaut *)
    	END_IF
    END_IF

    c_ready_old := c_ready;

    (* Der Datenempfang wird angehalten solange ein Sendevorgang läuft *)
    (* sonst kann es vorkommen das die Antwort-daten schon empfangen werden, *)
    (* bevor der Sendevorgang vom programm abgeschlossen wurde *)

    IF c_ready AND NOT s_active AND IP_C.MAILBOX[3] = 0 THEN
    	IF R_BUF.SIZE >= INT_TO_UINT(r_max_size) THEN
    		R_BUF.SIZE := UINT#0;
    		r_status := 254; (* Empfangsbuffer wegen Überlauf rückgesetzt *)
    	END_IF

    	r_offset := SEL(udp_mode,UINT_TO_INT(R_BUF.SIZE),0);
    	r_count := r_max_size - r_offset;

    	IF udp_mode THEN
    		bytes_received := SysSockRecvFrom(socket, ADR(R_BUF.BUFFER), r_count, 0, ADR(sockaddr), SIZEOF(sockaddr));

    		IF c_mode = BYTE#3 AND sockaddr.sin_addr <> SysSockNtohl(c_ip) THEN (* Mode 3 = UDP + PASSIVE + PORT + IP  auf richtige Partner-IP prüfen *)
    			bytes_received := 0;
    			R_BUF.SIZE := UINT#0;
    			sockaddr.sin_port := SysSockNtohs(c_port);
    			sockaddr.sin_addr := SysSockNtohl(c_ip);
    		END_IF

    	ELSE
    		bytes_received := SysSockRecv(socket, ADR(R_BUF.BUFFER[r_offset]), r_count, 0);
    	END_IF

    	(*UDP: IPC returns -1 if no data available or error occured,841 returns -1 if error occured and 0 if no data available*)
    	CASE bytes_received OF
    	-2147483648..-1: ; (* No data available or error occured *)
    	 0: IF NOT udp_mode THEN (* TCP-Mode: socket wurde von remote geschlossen *)
    			c_status := 253;
    			c_ready := FALSE;
    		END_IF
    	ELSE (* daten wurden empfangen *)
      		r_time := tx; (* Receive Timer ruecksetzen *)
    		R_BUF.SIZE := INT_TO_UINT(r_offset + DINT_TO_UINT(bytes_received)); (* aktuelle buffersize eintragen *)
    		IP_C.MAILBOX[1] := IP_C.MAILBOX[1] + 1; (* Receive Info *)
    		IF IP_C.MAILBOX[1] = 0 THEN IP_C.MAILBOX[1] := 1; END_IF

    		(* ---------------------- Debug-Message ----------------------------*)
    		(*IF _debug_enable THEN
    			LOG_CL.NEW_MSG := 'IP_REC DATA: POS: ~1 : SIZE: ~2 TOTAL ~3 -IP_ID ~6';
    			LOG_CL.PRINTF[1] := INT_TO_STRING(r_offset);
    			LOG_CL.PRINTF[2] := INT_TO_STRING(r_count);
    			LOG_CL.PRINTF[3] := UINT_TO_STRING(R_BUF.SIZE);
    			LOG_CL.PRINTF[6] := INT_TO_STRING(debug_ID);
    			LOG_MSG();
    		END_IF*)
    		(* -----------------------------------------------------------------------------*)

    	END_CASE
    END_IF

    (* ---------------------------------------------- *)

    IF S_BUF.SIZE > 0 THEN
    	IF c_ready AND c_enable THEN
    		IF NOT s_active AND IP_C.MAILBOX[2] = 0 THEN
    			(* Gesamtanzahl an Bytes limitieren und uebergeben *)
    			s_total := LIMIT(0,UINT_TO_INT(S_BUF.SIZE),r_max_size);
    			s_cur_pos  := 0;
    			s_cur_size := 0;
    			s_start := TRUE; (* Daten kopieren und senden anstossen *)
    			s_active := TRUE; (* Sende-Betrieb aktivieren *)
    			(* ---------------------- Debug-Message ----------------------------*)
    			(*IF _debug_enable THEN
    				LOG_CL.NEW_MSG := 'IP_SEN INIT: TOTAL: ~1 -IP_ID ~6';
    				LOG_CL.PRINTF[1] := INT_TO_STRING(s_total);
    				LOG_CL.PRINTF[6] := INT_TO_STRING(debug_ID);
    				LOG_MSG();
    			END_IF*)
    			(* -----------------------------------------------------------------------------*)
    		END_IF

    		IF s_done OR s_start THEN (* Daten senden aktiv *)

    			s_start := FALSE;
    			s_cur_pos := s_cur_pos + s_cur_size; (* neue Sende-Datenposition bestimmen *)
    			IF s_total > s_cur_pos THEN (* weitere Daten zum senden vorhanden ? *)
    				s_cur_size := s_total - s_cur_pos;
    				s_cur_size := LIMIT(0, s_cur_size, s_max_size); (* Telegrammlänge begrenzen *)

    				(* ---------------------- Debug-Message ----------------------------*)
    				(*IF _debug_enable THEN
    					LOG_CL.NEW_MSG := 'IP_SEN DATA: POS: ~1 : SIZE: ~2 TOTAL ~3 -IP_ID ~6';
    					LOG_CL.PRINTF[1] := INT_TO_STRING(s_cur_pos);
    					LOG_CL.PRINTF[2] := INT_TO_STRING(s_cur_size);
    					LOG_CL.PRINTF[3] := INT_TO_STRING(s_total);
    					LOG_CL.PRINTF[6] := INT_TO_STRING(debug_ID);
    					LOG_MSG();
    				END_IF*)
    				(* -----------------------------------------------------------------------------*)

    				s_time := tx; (* Send Timer ruecksetzen *)
    				r_time := tx; (* Receive Timer ruecksetzen *)
    				s_req := TRUE;

    			ELSE
    				(* keine weitere Sendedaten vorhanden -> Senden beenden *)
    				s_req := FALSE;
    				s_active := FALSE;
    				S_BUF.SIZE := 0;
    				(* ---------------------- Debug-Message ----------------------------*)
    				(*IF _debug_enable THEN
    					LOG_CL.NEW_MSG := 'IP_SEN FINISH -IP_ID ~6';
    					LOG_CL.PRINTF[6] := INT_TO_STRING(debug_ID);
    					LOG_MSG();
    				END_IF*)
    				(* -----------------------------------------------------------------------------*)
    			END_IF
    		END_IF
    	END_IF
    END_IF

    IF s_req THEN
    	s_done := FALSE;
    	IF udp_mode THEN
    		bytes_sent := SysSockSendTo(socket, ADR(S_BUF.BUFFER[s_cur_pos]), s_cur_size, 0, ADR(sockaddr), SIZEOF(sockaddr));
    	ELSE
    		bytes_sent := SysSockSend(socket, ADR(S_BUF.BUFFER[s_cur_pos]), s_cur_size, 0);
    	END_IF

    	CASE bytes_sent OF
    	-2147483648..-1:	; (* ERROR: Noch nicht bereit um Daten aufzunehmen -> nächsten Zyklus wieder probieren *)
    	 0: IF NOT udp_mode THEN (* TCP-Mode: socket wurde von remote geschlossen *)
    			c_status := 253;
    			c_ready := FALSE;
    		END_IF
    	ELSE
    		s_done := TRUE;
    		s_cur_size := DINT_TO_INT(bytes_sent); (* Anzahl der wirklich versendeten Bytes übernehmen *)
    		(* ---------------------- Debug-Message ----------------------------*)
    		(*IF _debug_enable THEN
    			LOG_CL.NEW_MSG := 'IP_SEN SEND_COUNT ~1 -IP_ID ~6';
    			LOG_CL.PRINTF[1] := DINT_TO_STRING(s_cur_size);
    			LOG_CL.PRINTF[6] := INT_TO_STRING(debug_ID);
    			LOG_MSG();
    		END_IF*)
    		(* -----------------------------------------------------------------------------*)
    	END_CASE
    END_IF

    (* ---------------------------------------------- *)

    IF IP_C.R_OBSERVE = FALSE OR s_active THEN
        r_time := tx;
    END_IF

    IF c_status = 0 AND tx - c_time > error_time AND c_enable AND NOT c_ready AND c_mode < 2 THEN (* Connect Timeout *)
    	c_status := 255; (* Timeout-Fehler ausgeben *)
    END_IF
    IF s_status = 0 AND tx - s_time > error_time AND s_active THEN (* Send Timeout *)
    	s_status := 255; (* Timeout-Fehler ausgeben *)
    END_IF
    IF r_status = 0 AND tx - r_time > error_time AND c_ready AND IP_C.R_OBSERVE THEN (* Receive Timeout *)
    	r_status := 255; (* Timeout-Fehler ausgeben *)
    END_IF

    IP_C.ERROR := DWORD_OF_BYTE(c_status,s_status,r_status,0);

    (* ---------------------- Debug-Message ----------------------------*)
    (*IF  _debug_enable THEN
    	IF (IP_C.ERROR <> debug_lasterror) THEN
    		LOG_CL.NEW_MSG := 'IP_ERROR ~1 -IP_ID ~6';
    		LOG_CL.PRINTF[1] := DWORD_TO_STRING(IP_C.ERROR);
    		LOG_CL.PRINTF[6] := INT_TO_STRING(debug_ID);
    		LOG_MSG();

    		debug_lasterror := IP_C.ERROR;
    		debug_last_id := debug_ID;
    	END_IF
    END_IF*)
    (* -----------------------------------------------------------------------------*)

    (* revision history
    ks	18. oct. 2008	rev 1.0
    	original version
    ks	05. jan. 2009	rev 1.1
    	zusätzlichen Parameter "PORT" hinzugefügt, und Code bei Verbindungsaufbau angepasst
    ks	28. feb. 2009	rev 1.2
    	connect code angepasst und verkürzung der zyklen bei Send
    ks	20. oct. 2009	rev 1.3
    	network_buffer basis 0
    ks	06. dec. 2009	rev 1.4
    	receive_count MAILBOX[1]
    ks	10. nov. 2010	rev 1.5
    	send_pause MAILBOX[2] and receive_pause MAILBOX[3]
    ks	07. feb. 2011	rev 1.6
    	Fehlercode 253 bei Remote-Verbindungsabbruch
    ks	30. may. 2011	rev 1.7
    	Fehler bei Empfangsüberwachung
    ks	26. july. 2011	rev 1.8
    	Error-Reset, diverse optimierungen
    ks	26. feb. 2012	rev 1.9
    	Code-Optimierung für höhere kompatibilität
    *)
END_FUNCTION_BLOCK

(* ---- IP_FIFO.st ---- *)
FUNCTION_BLOCK IP_FIFO
    (*http://www.oscat.de/images/OSCATNetwork/oscat_netlib121_en.pdf#page=108*)
    IF NOT FIFO.INIT THEN
    	FIFO.INIT := TRUE;
    	FIFO.NW := 1;
    	FIFO.NR := 1;
    	FIFO.EMPTY := TRUE;
    	FIFO.FULL := FALSE;
    	FIFO.TOP := 128; (* Arraygroesse 1 bis x *)
    	FIFO.MAX_ID := BYTE#1; (* maximale anzahl von Anmeldungen einer ID *)
    END_IF

    (* wenn keine ID vorhanden dann die naechste freie ID zuteilen *)
    IF ID = BYTE#00 THEN
    	IF FIFO.ID < INT_TO_BYTE(FIFO.TOP) THEN
    		ID := USINT_TO_BYTE(BYTE_TO_USINT(FIFO.ID) + USINT#1); (* ID +1 *)
    		FIFO.ID := ID; (* ID eintragen *)
    	    	(*####################  DEBUG-MESSAGE  ###################################*)
    	    	(*IF _debug_enable THEN
    	      		LOG_CL.NEW_MSG := 'FIFO: NEW ID:~1';
    	      		LOG_CL.PRINTF[1]  := BYTE_TO_STRING(ID);
    	      		LOG_MSG();
    	    	END_IF*)
    	    	(*########################################################################*)
    	ELSIF STATE < BYTE#200 THEN
    		(*####################  DEBUG-MESSAGE  ###################################*)
    		(*IF _debug_enable THEN
    			LOG_CL.NEW_MSG := 'FIFO: OVERFLOW ADD ID';
    			LOG_MSG();
    		END_IF*)
    		(*########################################################################*)

    		(* sollte nie passieren ! -> es sind zuviele teilnehmer angemeldet *)
    		(* es wird keine Nummer vergeben und alle anfragen werden negativ beantwortet *)
    		STATE := BYTE#255;
    		RETURN;
    	END_IF
    END_IF

    IF STATE = BYTE#1 AND NOT FIFO.FULL THEN (* Anmelden *)
    	(* nur eintragen wenn maximale anzahl nicht ueberschritten wurde *)
    	tmp := BYTE_TO_INT(ID);
    	IF FIFO.Y[tmp] < FIFO.MAX_ID THEN
    		FIFO.Y[tmp] := USINT_TO_BYTE(BYTE_TO_USINT(FIFO.Y[tmp]) + USINT#1); (* IP_ID Zähler +1 *)
    		tmp := FIFO.NW; (* geht bei mir leider nicht anders *)
    		FIFO.X[tmp] := ID;
    		IF FIFO.NW = FIFO.TOP THEN FIFO.NW := 1; ELSE FIFO.NW := FIFO.NW + 1; END_IF
    		FIFO.FULL := FIFO.NW = FIFO.NR;
    		FIFO.EMPTY := FALSE;
    		STATE := BYTE#2; (* weiterschalten auf "Warten auf Freigabe" *)
    		(*####################  DEBUG-MESSAGE  ###################################*)
    		(*IF _debug_enable THEN
    			LOG_CL.NEW_MSG := 'FIFO: ADD ID:~1';
    			LOG_CL.PRINTF[1]  := BYTE_TO_STRING(ID);
    			LOG_MSG();
    		END_IF*)
    		(*########################################################################*)

    	END_IF
    END_IF

    IF STATE = BYTE#2 AND NOT FIFO.EMPTY THEN (* check current stack element *)
    	tmp := FIFO.NR; (* geht bei mir leider nicht anders *)
    	IF ID = FIFO.X[tmp] THEN
    	STATE := BYTE#3; (* weiterschalten auf "Zugriffsfreigabe" *)
    	END_IF
    END_IF

    IF STATE = BYTE#4 AND NOT FIFO.EMPTY THEN (* remove from stack *)
    	tmp := FIFO.NR; (* geht bei mir leider nicht anders *)
    	IF ID = FIFO.X[tmp] THEN
    		tmp := BYTE_TO_INT(ID); (* geht bei mir leider nicht anders *)
    		FIFO.Y[tmp] := USINT_TO_BYTE(BYTE_TO_USINT(FIFO.Y[tmp]) - USINT#1); (* ID Zähler -1 *)
    		IF FIFO.NR = FIFO.TOP THEN FIFO.NR := 1; ELSE FIFO.NR := FIFO.NR + 1; END_IF
    		FIFO.EMPTY := FIFO.NR = FIFO.NW;
    		FIFO.FULL := FALSE;
    		(*####################  DEBUG-MESSAGE  ###################################*)
    		(*IF _debug_enable THEN
    			LOG_CL.NEW_MSG := 'FIFO: REMOVE ID:~1';
    			LOG_CL.PRINTF[1]  := BYTE_TO_STRING(ID);
    			LOG_MSG();
    		END_IF*)
    		(*########################################################################*)
    	END_IF
    	STATE := BYTE#5; (* "Remove done" *)
    END_IF

    (* revision history
    ks	18. oct. 2008	rev 1.0
    	original version

    *)
END_FUNCTION_BLOCK

(* ---- IRTRANS_DECODE.st ---- *)
FUNCTION_BLOCK IRTRANS_DECODE
    (*http://www.oscat.de/images/OSCATNetwork/oscat_netlib121_en.pdf#page=36*)
    size := R_BUF.size;

    (* do nothing if the buffer is empty *)
    IF size > 0 AND IP_C.MAILBOX[1] <> z THEN
    	i := 0;
    	ERROR := TRUE;
    	stop := size - 2;
    	(* read characters before first comma and store in device *)
    	pt := ADR(DEV);
    	buffer := ADR(R_BUF.buffer);
    	WHILE i < stop DO
    		IF buffer[i] = 44 THEN EXIT; END_IF
    		pt := buffer[i];
    		pt := pt + 1;
    		i := i + 1;
    	END_WHILE
    	(* terminate the device string *)
    	pt := 0;
    	(* read after first comma and store in KEY *)
    	i := i + 1;
    	pt := ADR(KEY);
    	WHILE i < stop DO
    		pt := buffer[i];
    		pt := pt + 1;
    		i := i + 1;
    	END_WHILE
    	(* terminate the KEY string *)
    	pt:= 0;
    	(* check if last two characters are $R$N 13, 10 *)
    	IF buffer[i] <> 13 AND buffer[i+1] <> 10 THEN	RETURN;	END_IF
    	(* check if device and KEY are present *)
    	IF LEN(DEV) = 0 OR LEN(KEY) = 0 THEN RETURN; END_IF
    	(* a valid transmission has been received *)
    	CMD := TRUE;
    	ERROR := FALSE;
    ELSE
    	ERROR := FALSE;
    	CMD := FALSE;
    END_IF

    z := IP_C.MAILBOX[1];

    (* revision history
    ks	18. oct. 2008	rev 1.0
    	original version
    ks	20. oct. 2009	rev 1.1
    	Networkbuffer und buffer-funktionen auf Basis 0
    ks	06. dec. 2009	rev 1.2
    	Codeanpassung für IRTRANS_SERVER
    *)
END_FUNCTION_BLOCK

(* ---- IRTRANS_RCV_1.st ---- *)
FUNCTION_BLOCK IRTRANS_RCV_1
    (*http://www.oscat.de/images/OSCATNetwork/oscat_netlib121_en.pdf#page=37*)
    Q := CMD AND DEV_CODE = DEV AND KEY_CODE = KEY;

    (* revision history
    hm	2. jan 2008		rev 1.0
    	original version

    hm	20. 6. 2008		rev 1.1
    	performance improvement

    hm	19. oct. 2008	rev 1.2
    	changed input device_code to DEV_CODE and device to DEV for compatibility reasons

    hm	06. dec. 2008	rev 1.3
    	IRTRANS_1 renamed to IRTRANS_RCV_1

    *)
END_FUNCTION_BLOCK

(* ---- IRTRANS_RCV_4.st ---- *)
FUNCTION_BLOCK IRTRANS_RCV_4
    (*http://www.oscat.de/images/OSCATNetwork/oscat_netlib121_en.pdf#page=39*)
    decode := CMD AND DEV_CODE = DEV;

    Q0 := KEY = KEY_CODE_0 AND decode;
    Q1 := KEY = KEY_CODE_1 AND decode;
    Q2 := KEY = KEY_CODE_2 AND decode;
    Q3 := KEY = KEY_CODE_3 AND decode;

    (* revision history
    hm	2. jan 2008		rev 1.0
    	original version

    hm	17. oct. 2008	rev 1.1
    	improved performance

    hm	19. oct. 2008	rev 1.2
    	changed input device_code to DEV_CODE and device to DEV for compatibility reasons

    hm	06. dec. 2008	rev 1.3
    	IRTRANS_1 renamed to IRTRANS_RCV_4

    *)
END_FUNCTION_BLOCK

(* ---- IRTRANS_RCV_8.st ---- *)
FUNCTION_BLOCK IRTRANS_RCV_8
    (*http://www.oscat.de/images/OSCATNetwork/oscat_netlib121_en.pdf#page=39*)
    decode := CMD AND DEV_CODE = DEV;

    Q0 := KEY = KEY_CODE_0 AND decode;
    Q1 := KEY = KEY_CODE_1 AND decode;
    Q2 := KEY = KEY_CODE_2 AND decode;
    Q3 := KEY = KEY_CODE_3 AND decode;
    Q4 := KEY = KEY_CODE_4 AND decode;
    Q5 := KEY = KEY_CODE_5 AND decode;
    Q6 := KEY = KEY_CODE_6 AND decode;
    Q7 := KEY = KEY_CODE_7 AND decode;

    (* revision history
    hm	2. jan 2008		rev 1.0
    	original version

    hm	17. oct 2008	rev 1.1
    	improved performance

    hm	19. oct. 2008	rev 1.2
    	changed input device_code to DEV_CODE and device to DEV for compatibility reasons

    hm	06. dec. 2008	rev 1.3
    	IRTRANS_1 renamed to IRTRANS_RCV_8

    *)
END_FUNCTION_BLOCK

(* ---- IRTRANS_SERVER.st ---- *)
FUNCTION_BLOCK IRTRANS_SERVER
    (*http://www.oscat.de/images/OSCATNetwork/oscat_netlib121_en.pdf#page=40*)
    IF NOT IP_C.C_ENABLE THEN
    	(* IP Datenverkehr einrichten *)
    	IP_C.C_PORT := WORD#0; (* Portnummer eintragen *)
    	IP_C.C_IP := DWORD#00; (* IP eintragen *)
    	IP_C.C_MODE := SEL(UDP_TCP,5,4); (* 4 = Mode: TCP+PASSIV+PORT / 5 = Mode: UDP+PASSIV+PORT*)
    	IP_C.C_ENABLE := TRUE; (* Verbindungsaufbau freigeben *)
    	IP_C.R_OBSERVE := FALSE; (* Datenempfang ueberwachen *)
    	IP_C.TIME_RESET := TRUE; (* Zeitueberwachung rücksetzen *)
    	S_BUF.SIZE := UINT#0; (* Sendedaten rücksetzen *)
    	R_BUF.SIZE := UINT#0; (* Empfangsdaten rücksetzen *)
    END_IF

    R_ENABLE := IP_C.C_STATE > 127;
    S_ENABLE := R_ENABLE AND (IP_C.MAILBOX[1] > 0 OR IP_C.C_MODE <> 5);
    ERROR := IP_C.ERROR;

    t(IN:= IP_C.ERROR > 0, PT:=t#5s);
    IF t.Q THEN
    	IP_C.TIME_RESET := TRUE; (* ERROR Reset *)
    END_IF

    (* revision history
    ks	6. dec 2009		rev 1.0
    	original version

    ks	17. may 2011		rev 1.1
    	neue Fehlerausgabe und Empfangsbuffer rücksetzen
    *)
END_FUNCTION_BLOCK

(* ---- IRTRANS_SND_1.st ---- *)
FUNCTION_BLOCK IRTRANS_SND_1
    (*http://www.oscat.de/images/OSCATNetwork/oscat_netlib121_en.pdf#page=42*)
    d := IP_C.C_STATE > 127 AND (IP_C.MAILBOX[1] > 0 OR IP_C.C_MODE <> 5);
    IF NOT d THEN RETURN; END_IF

    t(IN:= lk = k , PT:=T_REPEAT);

    IF S_BUF.size = 0 THEN
    	IF IN THEN
    		skey := KEY_CODE; k := 1;
    	ELSE
    		lk := 0;
    		KEY := 0;
    		RETURN; (* beenden wenn kein KEY aktiv *)
    	END_IF

    	IF lk <> k OR t.Q THEN (* anderer KEY oder repeat wartezeit abgelaufen *)
    		str := CONCAT('snd ',DEV_CODE);
    		str := CONCAT(str,',');
    		str := CONCAT(str,skey);
    		size := LEN(str);
    		_STRING_TO_BUFFER(str:=str, POS:=0, PT:=ADR(S_BUF.BUFFER), size:=size);
    		S_BUF.size := size; (* Sendelänge eintragen *)
    		KEY := k;
    		lk := k; (* letzten KEY speichern *)
    		t(IN:=FALSE); (* Reset Time *)
    	END_IF
    END_IF

    (* revision history
    hm	6. dec 2009		rev 1.0
    	original version
    *)
END_FUNCTION_BLOCK

(* ---- IRTRANS_SND_4.st ---- *)
FUNCTION_BLOCK IRTRANS_SND_4
    (*http://www.oscat.de/images/OSCATNetwork/oscat_netlib121_en.pdf#page=43*)
    d := IP_C.C_STATE > 127 AND (IP_C.MAILBOX[1] > 0 OR IP_C.C_MODE <> 5);
    IF NOT d THEN RETURN; END_IF

    t(IN:= lk = k , PT:=T_REPEAT);

    IF S_BUF.size = 0 THEN
    	IF IN_0 THEN
    		skey := KEY_CODE_0; k := 1;
    	ELSIF IN_1 THEN
    		skey := KEY_CODE_1; k := 2;
    	ELSIF IN_2 THEN
    		skey := KEY_CODE_2; k := 3;
    	ELSIF IN_3 THEN
    		skey := KEY_CODE_3; k := 4;
    	ELSE
    		lk := 0;
    		KEY := 0;
    		RETURN; (* beenden wenn kein KEY aktiv *)
    	END_IF

    	IF lk <> k OR t.Q THEN (* anderer KEY oder repeat wartezeit abgelaufen *)
    		str := CONCAT('snd ',DEV_CODE);
    		str := CONCAT(str,',');
    		str := CONCAT(str,skey);
    		size := LEN(str);
    		_STRING_TO_BUFFER(str:=str, POS:=0, PT:=ADR(S_BUF.BUFFER), size:=size);
    		S_BUF.size := size; (* Sendelänge eintragen *)
    		KEY := k;
    		lk := k; (* letzten KEY speichern *)
    		t(IN:=FALSE); (* Reset Time *)
    	END_IF
    END_IF

    (* revision history
    hm	6. dec 2009		rev 1.0
    	original version
    *)
END_FUNCTION_BLOCK

(* ---- IRTRANS_SND_8.st ---- *)
FUNCTION_BLOCK IRTRANS_SND_8
    (*http://www.oscat.de/images/OSCATNetwork/oscat_netlib121_en.pdf#page=44*)
    d := IP_C.C_STATE > 127 AND (IP_C.MAILBOX[1] > 0 OR IP_C.C_MODE <> 5);
    IF NOT d THEN RETURN; END_IF

    t(IN:= lk = k , PT:=T_REPEAT);

    IF S_BUF.size = 0 THEN
    	IF IN_0 THEN
    		skey := KEY_CODE_0; k := 1;
    	ELSIF IN_1 THEN
    		skey := KEY_CODE_1; k := 2;
    	ELSIF IN_2 THEN
    		skey := KEY_CODE_2; k := 3;
    	ELSIF IN_3 THEN
    		skey := KEY_CODE_3; k := 4;
    	ELSIF IN_4 THEN
    		skey := KEY_CODE_4; k := 5;
    	ELSIF IN_5 THEN
    		skey := KEY_CODE_5; k := 6;
    	ELSIF IN_6 THEN
    		skey := KEY_CODE_6; k := 7;
    	ELSIF IN_7 THEN
    		skey := KEY_CODE_7; k := 8;
    	ELSE
    		lk := 0;
    		KEY := 0;
    		RETURN; (* beenden wenn kein KEY aktiv *)
    	END_IF

    	IF lk <> k OR t.Q THEN (* anderer KEY oder repeat wartezeit abgelaufen *)
    		str := CONCAT('snd ',DEV_CODE);
    		str := CONCAT(str,',');
    		str := CONCAT(str,skey);
    		size := LEN(str);
    		_STRING_TO_BUFFER(str:=str, POS:=0, PT:=ADR(S_BUF.BUFFER), size:=size);
    		S_BUF.size := size; (* Sendelänge eintragen *)
    		KEY := k;
    		lk := k; (* letzten KEY speichern *)
    		t(IN:=FALSE); (* Reset Time *)
    	END_IF
    END_IF

    (* revision history
    hm	6. dec 2009		rev 1.0
    	original version
    *)
END_FUNCTION_BLOCK

(* ---- LOG_MSG.st ---- *)
FUNCTION_BLOCK LOG_MSG
    (*http://www.oscat.de/images/OSCATNetwork/oscat_netlib121_en.pdf#page=111*)
    IF DWORD_TO_BYTE(SHL(LOG_CL.NEW_MSG_OPTION,16)) > LOG_CL.LEVEL THEN RETURN; END_IF (* Logging freigegeben ?*)

    FB_PRINT_SF(PRINTF_DATA := LOG_CL.PRINTF,STR := LOG_CL.NEW_MSG);

    IF LOG_CL.RESET THEN (* Logeinträge löschen *)
    	LOG_CL.RESET := FALSE;
    	LOG_CL.RING_MODE := FALSE;
    	LOG_CL.idX := 0;
    	LOG_CL.UPDATE_COUNT := LOG_CL.UPDATE_COUNT + UINT#1; (* UpdateCount erhöhen *)
    END_IF

    IF LOG_CL.SIZE > 0 THEN (* size wert ist eingetragen *)
    	IF LEN(LOG_CL.NEW_MSG) > 0 THEN (* Meldung in Puffer eintragen *)
    		IF (LOG_CL.idX >= LOG_CL.SIZE) THEN
    			LOG_CL.RING_MODE := TRUE; (* bei Überlauf = Ringbuffermodus *)
    			LOG_CL.idX := 0; (* wieder auf arrayanfang positionieren *)
    		END_IF

    		LOG_CL.UPDATE_COUNT := LOG_CL.UPDATE_COUNT + UINT#1; (* UpdateCount erhöhen *)
    		LOG_CL.idX := LOG_CL.idX + INT#1; (* nächste freie Position *)
    		idX := LOG_CL.idX; (* lade aktuelle Log-Puffer Positition *)
    		LOG_CL.MSG[idX] := LOG_CL.NEW_MSG; (* neuen Log-String in puffer ablegen  *)
    		LOG_CL.MSG_OPTION[idX] := LOG_CL.NEW_MSG_OPTION; (* neue Log-String Option in puffer ablegen  *)
    		LOG_CL.NEW_MSG := ''; (* letzten Log-String löschen *)
    	END_IF
    END_IF
END_FUNCTION_BLOCK

(* ---- LOG_VIEWPORT.st ---- *)
FUNCTION_BLOCK LOG_VIEWPORT
    (*http://www.oscat.de/images/OSCATNetwork/oscat_netlib121_en.pdf#page=111*)
    (* Scroll Button verarbeiten *)
    IF LV.MOVE_TO_X <> 0 THEN
    	CASE LV.MOVE_TO_X OF
    	30000: pos := 1 ; (* älteste Meldung anzeigen *)
    	30001: pos := LC.SIZE; (* neueste Meldung anzeigen *)
    	30002: pos := pos + LV.count; (* eine Seite nach unten blättern -> Richtung neuere Nachrichten *)
    	30003: pos := pos - LV.count; (* eine Seite nach oben blättern -> Richtung ältere Nachrichten *)
    	ELSE
    		pos := pos + LV.MOVE_TO_X;
    	END_CASE
    	update_pos := TRUE;
    	LV.MOVE_TO_X := 0;
    END_IF

    IF (LV.UPDATE_COUNT <> LC.UPDATE_COUNT) OR update_pos THEN (* Aktualisierung überwachen *)
    	LV.UPDATE := TRUE;
    	LV.UPDATE_COUNT := LC.UPDATE_COUNT;
    	update_pos := FALSE;

    	(* pos prüfen und übernehmen *)
    	IF LC.RING_MODE THEN
    		pos := LIMIT(1,pos,LC.SIZE - LV.count + 1);
    	ELSE
    		IF LC.idx > LV.count THEN
    			pos := LIMIT(1,pos,LC.idx - LV.count + 1);
    		ELSE
    			pos := 1;
    		END_IF
    	END_IF

    	(* idxBasis berechnen *)
    	base := LC.idx - pos - LV.count + 1;
    	IF LC.RING_MODE THEN
    		(* Anzeige im Ringpuffermodus *)
    		FOR count:= 1 TO LV.count DO
    			idx := base + count;
    			IF idx < 1 THEN
    				idx := idx + LC.SIZE;
    			END_IF
    			LV.LINE_ARRAY[count] := idx;
    		END_FOR
    	ELSE
    		(* Anzeige im Normalmodus *)
    		FOR count:= 1 TO LV.count DO
    			idx := base + count;
    			IF idx < 1 THEN
    				(* Leere Zeile ausgeben *)
    				LV.LINE_ARRAY[count] := 0;
    			ELSE
    				LV.LINE_ARRAY[count] := idx;
    			END_IF
    		END_FOR
    	END_IF
    END_IF

    (* revision history
    ks	01. mai 2010	rev 1.0
    	original version

    ks	05. mai 2012	rev 1.1
    	Fehler im Ringmodus

    *)
END_FUNCTION_BLOCK
